Yaskawa INFORM job: A_ROOF_UPPER_0614_2_PAINT_46.JBI

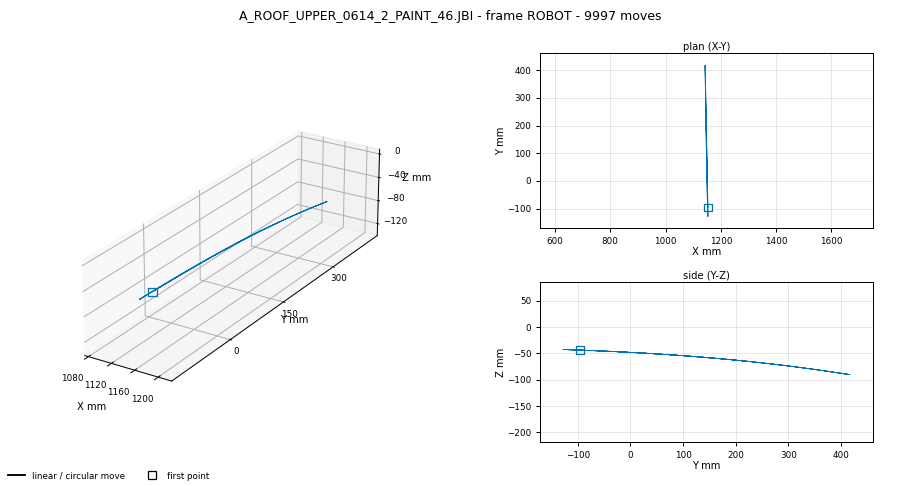
[picture p0: tool path of A_ROOF_UPPER_0614_2_PAINT_46.JBI in frame ROBOT, 9997 of 9997 moves have a stored position in this frame; points joined in program order, loops and branches not executed]
/JOB
//NAME A_ROOF_UPPER_0614_2_PAINT46
//POS
///NPOS 9997,0,0,0,0,0
///TOOL 1
///USER 0
///POSTYPE ROBOT
///RECTAN
///RCONF 1,0,0,0,0,0,0,0,0,0,0,0,0,0,0,0,0,0,0,0,0,0,0,0
C00000=1153.348,-96.269,-43.440,178.853,5.937,149.402
C00001=1153.343,-96.020,-43.449,178.855,5.937,149.401
C00002=1153.337,-95.770,-43.459,178.857,5.937,149.401
C00003=1153.332,-95.520,-43.468,178.859,5.937,149.400
C00004=1153.326,-95.270,-43.478,178.861,5.938,149.400
C00005=1153.321,-95.020,-43.487,178.863,5.939,149.399
C00006=1153.315,-94.771,-43.497,178.865,5.939,149.399
C00007=1153.310,-94.521,-43.506,178.867,5.939,149.398
C00008=1153.304,-94.271,-43.515,178.870,5.940,149.398
C00009=1153.299,-94.021,-43.525,178.871,5.940,149.397
C00010=1153.294,-93.772,-43.534,178.874,5.940,149.396
C00011=1153.289,-93.522,-43.544,178.876,5.941,149.396
C00012=1153.283,-93.272,-43.553,178.878,5.941,149.395
C00013=1153.278,-93.023,-43.563,178.880,5.942,149.395
C00014=1153.273,-92.773,-43.572,178.882,5.941,149.394
C00015=1153.267,-92.523,-43.582,178.884,5.942,149.394
C00016=1153.262,-92.273,-43.592,178.886,5.943,149.393
C00017=1153.257,-92.023,-43.602,178.888,5.942,149.393
C00018=1153.252,-91.773,-43.611,178.891,5.943,149.392
C00019=1153.246,-91.524,-43.621,178.893,5.944,149.392
C00020=1153.241,-91.274,-43.630,178.895,5.943,149.391
C00021=1153.235,-91.024,-43.640,178.897,5.944,149.390
C00022=1153.230,-90.775,-43.649,178.899,5.945,149.390
C00023=1153.225,-90.525,-43.659,178.901,5.945,149.389
C00024=1153.219,-90.275,-43.668,178.904,5.945,149.389
C00025=1153.214,-90.026,-43.678,178.906,5.946,149.388
C00026=1153.209,-89.775,-43.687,178.907,5.946,149.388
C00027=1153.204,-89.526,-43.698,178.910,5.946,149.387
C00028=1153.198,-89.276,-43.707,178.912,5.947,149.387
C00029=1153.193,-89.026,-43.717,178.914,5.947,149.386
C00030=1153.188,-88.777,-43.726,178.917,5.947,149.385
C00031=1153.182,-88.527,-43.736,178.919,5.948,149.385
C00032=1153.176,-88.277,-43.746,178.920,5.948,149.384
C00033=1153.171,-88.027,-43.755,178.923,5.949,149.384
C00034=1153.166,-87.777,-43.766,178.925,5.949,149.383
C00035=1153.161,-87.528,-43.775,178.927,5.949,149.383
C00036=1153.156,-87.278,-43.785,178.929,5.950,149.382
C00037=1153.151,-87.028,-43.794,178.932,5.950,149.382
C00038=1153.145,-86.779,-43.804,178.933,5.950,149.381
C00039=1153.139,-86.529,-43.814,178.935,5.951,149.381
C00040=1153.135,-86.279,-43.824,178.938,5.952,149.380
C00041=1153.129,-86.029,-43.833,178.940,5.952,149.379
C00042=1153.124,-85.779,-43.843,178.942,5.952,149.379
C00043=1153.119,-85.530,-43.853,178.945,5.953,149.378
C00044=1153.113,-85.280,-43.863,178.946,5.953,149.378
C00045=1153.108,-85.031,-43.872,178.948,5.953,149.377
C00046=1153.103,-84.780,-43.883,178.951,5.954,149.377
C00047=1153.098,-84.531,-43.893,178.953,5.954,149.376
C00048=1153.092,-84.281,-43.902,178.955,5.955,149.376
C00049=1153.086,-84.031,-43.912,178.957,5.955,149.375
C00050=1153.082,-83.782,-43.922,178.959,5.955,149.374
C00051=1153.076,-83.531,-43.932,178.961,5.956,149.374
C00052=1153.071,-83.282,-43.942,178.964,5.956,149.373
C00053=1153.066,-83.032,-43.952,178.966,5.956,149.373
C00054=1153.060,-82.783,-43.962,178.968,5.957,149.372
C00055=1153.054,-82.533,-43.971,178.970,5.957,149.372
C00056=1153.050,-82.283,-43.981,178.972,5.957,149.371
C00057=1153.044,-82.033,-43.991,178.974,5.958,149.371
C00058=1153.039,-81.784,-44.002,178.977,5.958,149.370
C00059=1153.034,-81.534,-44.011,178.978,5.958,149.369
C00060=1153.029,-81.284,-44.021,178.981,5.959,149.369
C00061=1153.023,-81.034,-44.031,178.983,5.959,149.368
C00062=1153.017,-80.785,-44.042,178.986,5.960,149.368
C00063=1153.013,-80.535,-44.051,178.987,5.960,149.367
C00064=1153.007,-80.284,-44.061,178.990,5.961,149.366
C00065=1153.002,-80.035,-44.071,178.992,5.961,149.366
C00066=1152.997,-79.786,-44.081,178.994,5.961,149.366
C00067=1152.991,-79.536,-44.091,178.996,5.962,149.365
C00068=1152.986,-79.286,-44.102,178.998,5.962,149.364
C00069=1152.981,-79.036,-44.112,179.000,5.962,149.364
C00070=1152.976,-78.786,-44.121,179.003,5.963,149.363
C00071=1152.970,-78.537,-44.131,179.005,5.964,149.363
C00072=1152.965,-78.287,-44.142,179.008,5.964,149.362
C00073=1152.959,-78.037,-44.152,179.009,5.964,149.361
C00074=1152.954,-77.788,-44.161,179.011,5.965,149.361
C00075=1152.949,-77.538,-44.172,179.014,5.965,149.360
C00076=1152.944,-77.288,-44.182,179.016,5.965,149.360
C00077=1152.938,-77.039,-44.192,179.018,5.966,149.359
C00078=1152.933,-76.767,-44.203,179.020,5.966,149.359
C00079=1152.926,-76.496,-44.214,179.023,5.967,149.358
C00080=1152.921,-76.224,-44.225,179.025,5.967,149.357
C00081=1152.915,-75.953,-44.236,179.028,5.968,149.357
C00082=1152.910,-75.703,-44.246,179.030,5.968,149.356
C00083=1152.905,-75.454,-44.256,179.032,5.969,149.356
C00084=1152.900,-75.204,-44.267,179.034,5.969,149.355
C00085=1152.894,-74.954,-44.277,179.037,5.970,149.355
C00086=1152.888,-74.705,-44.287,179.038,5.970,149.354
C00087=1152.883,-74.455,-44.298,179.041,5.970,149.353
C00088=1152.878,-74.205,-44.308,179.043,5.971,149.353
C00089=1152.872,-73.955,-44.318,179.045,5.971,149.352
C00090=1152.867,-73.706,-44.328,179.047,5.971,149.352
C00091=1152.862,-73.456,-44.338,179.050,5.972,149.351
C00092=1152.857,-73.206,-44.348,179.052,5.972,149.350
C00093=1152.852,-72.956,-44.359,179.054,5.972,149.350
C00094=1152.846,-72.707,-44.369,179.056,5.973,149.350
C00095=1152.841,-72.457,-44.379,179.059,5.974,149.349
C00096=1152.836,-72.207,-44.390,179.061,5.974,149.348
C00097=1152.830,-71.957,-44.400,179.062,5.974,149.348
C00098=1152.825,-71.708,-44.410,179.065,5.975,149.347
C00099=1152.820,-71.458,-44.420,179.067,5.975,149.347
C00100=1152.815,-71.208,-44.431,179.070,5.976,149.346
C00101=1152.809,-70.959,-44.441,179.072,5.976,149.345
C00102=1152.804,-70.708,-44.451,179.074,5.977,149.345
C00103=1152.798,-70.459,-44.462,179.076,5.977,149.344
C00104=1152.793,-70.209,-44.472,179.079,5.978,149.344
C00105=1152.788,-69.960,-44.483,179.080,5.978,149.343
C00106=1152.783,-69.710,-44.493,179.083,5.978,149.343
C00107=1152.778,-69.460,-44.504,179.085,5.979,149.342
C00108=1152.772,-69.210,-44.514,179.088,5.979,149.341
C00109=1152.766,-68.961,-44.524,179.089,5.979,149.341
C00110=1152.761,-68.711,-44.535,179.092,5.980,149.340
C00111=1152.756,-68.461,-44.545,179.094,5.980,149.340
C00112=1152.751,-68.211,-44.556,179.096,5.981,149.339
C00113=1152.745,-67.962,-44.567,179.098,5.981,149.339
C00114=1152.741,-67.713,-44.576,179.101,5.982,149.338
C00115=1152.736,-67.462,-44.587,179.103,5.982,149.338
C00116=1152.730,-67.213,-44.597,179.106,5.983,149.337
C00117=1152.725,-66.963,-44.608,179.107,5.983,149.336
C00118=1152.719,-66.713,-44.618,179.109,5.984,149.336
C00119=1152.715,-66.463,-44.629,179.112,5.984,149.335
C00120=1152.709,-66.214,-44.639,179.114,5.985,149.335
C00121=1152.703,-65.964,-44.649,179.116,5.984,149.334
C00122=1152.698,-65.714,-44.660,179.118,5.985,149.334
C00123=1152.693,-65.465,-44.671,179.121,5.986,149.333
C00124=1152.687,-65.215,-44.682,179.123,5.986,149.332
C00125=1152.682,-64.965,-44.692,179.126,5.987,149.332
C00126=1152.677,-64.715,-44.703,179.128,5.987,149.331
C00127=1152.672,-64.466,-44.714,179.130,5.987,149.331
C00128=1152.667,-64.216,-44.724,179.132,5.988,149.330
C00129=1152.661,-63.966,-44.735,179.135,5.989,149.330
C00130=1152.656,-63.716,-44.745,179.136,5.989,149.329
C00131=1152.651,-63.467,-44.756,179.139,5.989,149.328
C00132=1152.646,-63.217,-44.767,179.141,5.990,149.328
C00133=1152.640,-62.967,-44.777,179.143,5.991,149.327
C00134=1152.635,-62.718,-44.788,179.146,5.991,149.327
C00135=1152.630,-62.468,-44.798,179.148,5.991,149.326
C00136=1152.625,-62.218,-44.809,179.150,5.991,149.326
C00137=1152.620,-61.969,-44.820,179.152,5.992,149.325
C00138=1152.615,-61.719,-44.830,179.155,5.993,149.325
C00139=1152.608,-61.469,-44.841,179.157,5.993,149.324
C00140=1152.603,-61.219,-44.853,179.159,5.993,149.323
C00141=1152.598,-60.970,-44.863,179.162,5.994,149.323
C00142=1152.593,-60.719,-44.873,179.164,5.994,149.322
C00143=1152.588,-60.470,-44.884,179.166,5.995,149.322
C00144=1152.583,-60.220,-44.895,179.169,5.996,149.321
C00145=1152.577,-59.971,-44.906,179.170,5.996,149.321
C00146=1152.572,-59.721,-44.916,179.173,5.996,149.320
C00147=1152.567,-59.472,-44.927,179.175,5.997,149.319
C00148=1152.561,-59.222,-44.938,179.177,5.998,149.319
C00149=1152.556,-58.972,-44.949,179.180,5.998,149.318
C00150=1152.551,-58.722,-44.960,179.181,5.998,149.318
C00151=1152.546,-58.472,-44.970,179.184,5.998,149.317
C00152=1152.541,-58.223,-44.981,179.186,5.999,149.316
C00153=1152.536,-57.973,-44.992,179.188,6.000,149.316
C00154=1152.529,-57.723,-45.003,179.191,6.000,149.315
C00155=1152.525,-57.473,-45.014,179.193,6.000,149.315
C00156=1152.519,-57.224,-45.024,179.195,6.001,149.314
C00157=1152.514,-56.974,-45.036,179.198,6.001,149.314
C00158=1152.509,-56.724,-45.046,179.200,6.002,149.313
C00159=1152.503,-56.475,-45.058,179.202,6.003,149.312
C00160=1152.498,-56.225,-45.068,179.204,6.003,149.312
C00161=1152.493,-55.976,-45.079,179.207,6.003,149.311
C00162=1152.488,-55.725,-45.090,179.209,6.004,149.311
C00163=1152.483,-55.477,-45.101,179.212,6.004,149.310
C00164=1152.477,-55.227,-45.113,179.214,6.005,149.310
C00165=1152.472,-54.976,-45.123,179.216,6.006,149.309
C00166=1152.467,-54.727,-45.134,179.218,6.005,149.308
C00167=1152.462,-54.477,-45.145,179.220,6.006,149.308
C00168=1152.457,-54.227,-45.157,179.223,6.007,149.307
C00169=1152.451,-53.978,-45.167,179.225,6.007,149.307
C00170=1152.446,-53.728,-45.178,179.228,6.008,149.306
C00171=1152.441,-53.479,-45.188,179.230,6.008,149.306
C00172=1152.435,-53.229,-45.200,179.232,6.008,149.305
C00173=1152.431,-52.979,-45.211,179.234,6.009,149.304
C00174=1152.425,-52.729,-45.222,179.236,6.010,149.304
C00175=1152.420,-52.479,-45.233,179.239,6.010,149.303
C00176=1152.415,-52.230,-45.245,179.241,6.011,149.303
C00177=1152.409,-51.980,-45.255,179.243,6.012,149.302
C00178=1152.405,-51.731,-45.266,179.245,6.011,149.302
C00179=1152.398,-51.481,-45.277,179.248,6.012,149.301
C00180=1152.394,-51.231,-45.288,179.250,6.012,149.300
C00181=1152.389,-50.982,-45.300,179.253,6.013,149.300
C00182=1152.383,-50.711,-45.312,179.255,6.014,149.299
C00183=1152.377,-50.440,-45.324,179.257,6.014,149.299
C00184=1152.371,-50.169,-45.336,179.260,6.015,149.298
C00185=1152.365,-49.899,-45.348,179.263,6.015,149.297
C00186=1152.361,-49.649,-45.359,179.265,6.016,149.297
C00187=1152.356,-49.400,-45.371,179.268,6.016,149.296
C00188=1152.350,-49.150,-45.381,179.270,6.017,149.296
C00189=1152.345,-48.900,-45.393,179.271,6.017,149.295
C00190=1152.339,-48.650,-45.405,179.274,6.018,149.294
C00191=1152.334,-48.401,-45.415,179.276,6.018,149.294
C00192=1152.329,-48.151,-45.426,179.279,6.019,149.293
C00193=1152.324,-47.901,-45.438,179.281,6.020,149.293
C00194=1152.319,-47.652,-45.449,179.284,6.020,149.292
C00195=1152.313,-47.402,-45.460,179.286,6.021,149.292
C00196=1152.308,-47.152,-45.471,179.288,6.022,149.291
C00197=1152.303,-46.903,-45.483,179.290,6.021,149.290
C00198=1152.297,-46.653,-45.494,179.292,6.022,149.290
C00199=1152.293,-46.404,-45.505,179.295,6.022,149.289
C00200=1152.287,-46.153,-45.517,179.297,6.023,149.289
C00201=1152.282,-45.904,-45.528,179.300,6.024,149.288
C00202=1152.276,-45.654,-45.539,179.302,6.024,149.288
C00203=1152.271,-45.405,-45.551,179.305,6.025,149.287
C00204=1152.266,-45.155,-45.563,179.307,6.025,149.286
C00205=1152.261,-44.906,-45.573,179.308,6.025,149.286
C00206=1152.256,-44.656,-45.584,179.311,6.026,149.285
C00207=1152.250,-44.406,-45.596,179.313,6.027,149.285
C00208=1152.246,-44.156,-45.607,179.316,6.027,149.284
C00209=1152.240,-43.906,-45.619,179.318,6.028,149.284
C00210=1152.235,-43.657,-45.630,179.321,6.028,149.283
C00211=1152.229,-43.407,-45.642,179.323,6.029,149.282
C00212=1152.225,-43.158,-45.653,179.326,6.029,149.282
C00213=1152.219,-42.908,-45.665,179.327,6.029,149.281
C00214=1152.214,-42.658,-45.675,179.329,6.030,149.281
C00215=1152.208,-42.408,-45.687,179.332,6.031,149.280
C00216=1152.204,-42.159,-45.698,179.334,6.031,149.280
C00217=1152.198,-41.909,-45.710,179.337,6.032,149.279
C00218=1152.193,-41.659,-45.722,179.339,6.033,149.278
C00219=1152.187,-41.410,-45.733,179.342,6.033,149.278
C00220=1152.182,-41.160,-45.745,179.344,6.034,149.277
C00221=1152.177,-40.910,-45.756,179.347,6.034,149.277
C00222=1152.172,-40.660,-45.768,179.349,6.035,149.276
C00223=1152.167,-40.411,-45.779,179.350,6.035,149.276
C00224=1152.161,-40.161,-45.791,179.353,6.035,149.275
C00225=1152.156,-39.912,-45.802,179.355,6.036,149.274
C00226=1152.151,-39.662,-45.814,179.358,6.037,149.274
C00227=1152.146,-39.412,-45.826,179.360,6.037,149.273
C00228=1152.141,-39.162,-45.837,179.363,6.038,149.273
C00229=1152.135,-38.913,-45.849,179.365,6.039,149.272
C00230=1152.130,-38.663,-45.860,179.368,6.039,149.271
C00231=1152.125,-38.413,-45.872,179.370,6.040,149.271
C00232=1152.119,-38.164,-45.884,179.372,6.041,149.270
C00233=1152.115,-37.914,-45.895,179.375,6.041,149.270
C00234=1152.109,-37.664,-45.907,179.377,6.042,149.269
C00235=1152.104,-37.414,-45.918,179.379,6.041,149.269
C00236=1152.099,-37.166,-45.931,179.381,6.042,149.268
C00237=1152.093,-36.916,-45.943,179.384,6.043,149.267
C00238=1152.089,-36.666,-45.954,179.386,6.043,149.267
C00239=1152.083,-36.416,-45.966,179.389,6.044,149.266
C00240=1152.078,-36.166,-45.978,179.391,6.045,149.266
C00241=1152.073,-35.917,-45.989,179.394,6.045,149.265
C00242=1152.068,-35.667,-46.001,179.396,6.046,149.265
C00243=1152.062,-35.417,-46.012,179.398,6.047,149.264
C00244=1152.057,-35.168,-46.024,179.401,6.047,149.263
C00245=1152.052,-34.919,-46.036,179.403,6.048,149.263
C00246=1152.046,-34.669,-46.048,179.405,6.048,149.262
C00247=1152.042,-34.419,-46.059,179.408,6.049,149.262
C00248=1152.036,-34.169,-46.071,179.410,6.050,149.261
C00249=1152.031,-33.919,-46.083,179.412,6.050,149.261
C00250=1152.025,-33.669,-46.095,179.415,6.050,149.260
C00251=1152.021,-33.420,-46.107,179.417,6.051,149.259
C00252=1152.016,-33.170,-46.119,179.419,6.051,149.259
C00253=1152.010,-32.920,-46.131,179.422,6.052,149.258
C00254=1152.005,-32.671,-46.142,179.424,6.053,149.258
C00255=1152.000,-32.422,-46.154,179.426,6.053,149.257
C00256=1151.994,-32.172,-46.166,179.429,6.054,149.257
C00257=1151.989,-31.922,-46.178,179.431,6.054,149.256
C00258=1151.984,-31.673,-46.189,179.433,6.055,149.255
C00259=1151.979,-31.423,-46.202,179.436,6.056,149.255
C00260=1151.974,-31.173,-46.214,179.438,6.056,149.254
C00261=1151.968,-30.923,-46.226,179.441,6.057,149.254
C00262=1151.964,-30.674,-46.237,179.443,6.058,149.253
C00263=1151.958,-30.424,-46.250,179.446,6.058,149.252
C00264=1151.953,-30.174,-46.262,179.448,6.059,149.252
C00265=1151.948,-29.925,-46.273,179.451,6.059,149.251
C00266=1151.942,-29.675,-46.286,179.453,6.060,149.251
C00267=1151.938,-29.426,-46.297,179.455,6.061,149.250
C00268=1151.932,-29.176,-46.309,179.458,6.061,149.250
C00269=1151.927,-28.926,-46.322,179.460,6.062,149.249
C00270=1151.922,-28.676,-46.334,179.463,6.062,149.248
C00271=1151.916,-28.426,-46.346,179.465,6.063,149.248
C00272=1151.911,-28.177,-46.358,179.467,6.064,149.247
C00273=1151.906,-27.928,-46.369,179.469,6.064,149.247
C00274=1151.901,-27.678,-46.381,179.472,6.064,149.246
C00275=1151.896,-27.428,-46.394,179.474,6.065,149.246
C00276=1151.891,-27.178,-46.406,179.476,6.065,149.245
C00277=1151.885,-26.929,-46.418,179.479,6.066,149.244
C00278=1151.880,-26.679,-46.430,179.481,6.067,149.244
C00279=1151.876,-26.430,-46.442,179.483,6.067,149.243
C00280=1151.870,-26.180,-46.454,179.486,6.068,149.243
C00281=1151.865,-25.930,-46.466,179.488,6.069,149.242
C00282=1151.860,-25.681,-46.479,179.490,6.069,149.242
C00283=1151.854,-25.431,-46.491,179.493,6.070,149.241
C00284=1151.849,-25.182,-46.503,179.495,6.071,149.240
C00285=1151.844,-24.932,-46.515,179.498,6.071,149.240
C00286=1151.839,-24.662,-46.529,179.501,6.071,149.239
C00287=1151.833,-24.392,-46.542,179.503,6.073,149.239
C00288=1151.827,-24.122,-46.554,179.506,6.073,149.238
C00289=1151.822,-23.852,-46.569,179.509,6.074,149.237
C00290=1151.816,-23.602,-46.580,179.511,6.075,149.237
C00291=1151.811,-23.353,-46.593,179.513,6.075,149.236
C00292=1151.806,-23.103,-46.605,179.516,6.076,149.236
C00293=1151.801,-22.853,-46.618,179.518,6.077,149.235
C00294=1151.795,-22.603,-46.629,179.521,6.077,149.234
C00295=1151.791,-22.354,-46.641,179.523,6.078,149.234
C00296=1151.785,-22.105,-46.653,179.525,6.078,149.233
C00297=1151.780,-21.855,-46.666,179.528,6.079,149.233
C00298=1151.775,-21.605,-46.678,179.530,6.080,149.232
C00299=1151.770,-21.355,-46.691,179.532,6.080,149.232
C00300=1151.765,-21.106,-46.703,179.535,6.081,149.231
C00301=1151.760,-20.856,-46.715,179.537,6.082,149.230
C00302=1151.755,-20.607,-46.728,179.540,6.082,149.230
C00303=1151.749,-20.357,-46.740,179.542,6.083,149.229
C00304=1151.744,-20.107,-46.752,179.545,6.083,149.229
C00305=1151.738,-19.858,-46.766,179.547,6.084,149.228
C00306=1151.733,-19.608,-46.777,179.550,6.084,149.227
C00307=1151.728,-19.359,-46.790,179.552,6.085,149.227
C00308=1151.723,-19.109,-46.803,179.554,6.086,149.226
C00309=1151.718,-18.859,-46.815,179.557,6.086,149.226
C00310=1151.712,-18.609,-46.827,179.559,6.087,149.225
C00311=1151.707,-18.360,-46.840,179.562,6.088,149.225
C00312=1151.702,-18.110,-46.852,179.564,6.088,149.224
C00313=1151.697,-17.861,-46.865,179.566,6.089,149.223
C00314=1151.692,-17.611,-46.877,179.569,6.090,149.223
C00315=1151.687,-17.361,-46.889,179.571,6.090,149.222
C00316=1151.682,-17.111,-46.902,179.573,6.091,149.222
C00317=1151.677,-16.862,-46.915,179.576,6.091,149.221
C00318=1151.671,-16.613,-46.927,179.579,6.093,149.221
C00319=1151.666,-16.363,-46.939,179.581,6.093,149.220
C00320=1151.661,-16.113,-46.953,179.584,6.094,149.219
C00321=1151.656,-15.863,-46.965,179.586,6.095,149.219
C00322=1151.651,-15.614,-46.978,179.589,6.095,149.218
C00323=1151.645,-15.364,-46.990,179.591,6.096,149.218
C00324=1151.640,-15.115,-47.002,179.593,6.097,149.217
C00325=1151.635,-14.865,-47.015,179.596,6.097,149.216
C00326=1151.630,-14.615,-47.028,179.598,6.098,149.216
C00327=1151.624,-14.366,-47.041,179.600,6.099,149.215
C00328=1151.619,-14.116,-47.054,179.603,6.099,149.215
C00329=1151.614,-13.866,-47.066,179.605,6.100,149.214
C00330=1151.609,-13.616,-47.079,179.608,6.100,149.214
C00331=1151.604,-13.367,-47.091,179.610,6.101,149.213
C00332=1151.599,-13.118,-47.104,179.613,6.102,149.212
C00333=1151.593,-12.868,-47.117,179.615,6.102,149.212
C00334=1151.589,-12.618,-47.130,179.618,6.103,149.211
C00335=1151.583,-12.368,-47.142,179.620,6.104,149.211
C00336=1151.578,-12.119,-47.154,179.622,6.104,149.210
C00337=1151.573,-11.870,-47.167,179.625,6.106,149.210
C00338=1151.568,-11.619,-47.181,179.628,6.106,149.209
C00339=1151.563,-11.370,-47.193,179.630,6.107,149.209
C00340=1151.558,-11.121,-47.206,179.633,6.107,149.208
C00341=1151.552,-10.871,-47.218,179.635,6.108,149.207
C00342=1151.548,-10.621,-47.231,179.637,6.109,149.207
C00343=1151.542,-10.372,-47.245,179.640,6.109,149.206
C00344=1151.537,-10.122,-47.257,179.642,6.110,149.205
C00345=1151.532,-9.873,-47.270,179.644,6.111,149.205
C00346=1151.527,-9.623,-47.283,179.647,6.111,149.205
C00347=1151.521,-9.373,-47.296,179.649,6.112,149.204
C00348=1151.516,-9.124,-47.308,179.652,6.113,149.203
C00349=1151.512,-8.874,-47.321,179.655,6.114,149.203
C00350=1151.507,-8.625,-47.334,179.657,6.115,149.202
C00351=1151.501,-8.375,-47.347,179.660,6.115,149.202
C00352=1151.496,-8.125,-47.360,179.662,6.116,149.201
C00353=1151.491,-7.876,-47.373,179.664,6.116,149.200
C00354=1151.485,-7.626,-47.386,179.667,6.117,149.200
C00355=1151.481,-7.376,-47.399,179.669,6.118,149.199
C00356=1151.476,-7.127,-47.412,179.671,6.118,149.199
C00357=1151.470,-6.877,-47.425,179.674,6.119,149.198
C00358=1151.465,-6.628,-47.437,179.676,6.120,149.198
C00359=1151.460,-6.378,-47.450,179.679,6.120,149.197
C00360=1151.454,-6.128,-47.464,179.682,6.122,149.196
C00361=1151.449,-5.879,-47.476,179.684,6.122,149.196
C00362=1151.445,-5.629,-47.489,179.687,6.123,149.195
C00363=1151.439,-5.380,-47.503,179.689,6.123,149.195
C00364=1151.435,-5.130,-47.516,179.691,6.124,149.194
C00365=1151.429,-4.880,-47.529,179.694,6.125,149.193
C00366=1151.424,-4.631,-47.542,179.696,6.125,149.193
C00367=1151.419,-4.381,-47.555,179.698,6.126,149.193
C00368=1151.413,-4.131,-47.568,179.701,6.127,149.192
C00369=1151.408,-3.882,-47.581,179.704,6.128,149.191
C00370=1151.404,-3.632,-47.594,179.706,6.129,149.191
C00371=1151.398,-3.383,-47.607,179.709,6.130,149.190
C00372=1151.393,-3.133,-47.620,179.711,6.130,149.190
C00373=1151.388,-2.883,-47.634,179.713,6.131,149.189
C00374=1151.382,-2.634,-47.646,179.716,6.131,149.188
C00375=1151.378,-2.384,-47.660,179.718,6.132,149.188
C00376=1151.372,-2.135,-47.673,179.721,6.133,149.187
C00377=1151.368,-1.885,-47.686,179.724,6.134,149.187
C00378=1151.362,-1.635,-47.699,179.726,6.135,149.186
C00379=1151.357,-1.386,-47.712,179.729,6.135,149.186
C00380=1151.352,-1.136,-47.726,179.731,6.136,149.185
C00381=1151.347,-0.887,-47.739,179.733,6.137,149.184
C00382=1151.342,-0.637,-47.752,179.736,6.137,149.184
C00383=1151.337,-0.388,-47.766,179.738,6.138,149.183
C00384=1151.331,-0.138,-47.779,179.741,6.138,149.183
C00385=1151.326,0.112,-47.792,179.744,6.140,149.182
C00386=1151.320,0.361,-47.805,179.746,6.140,149.181
C00387=1151.316,0.611,-47.819,179.748,6.141,149.181
C00388=1151.310,0.860,-47.832,179.751,6.142,149.181
C00389=1151.306,1.110,-47.845,179.753,6.142,149.180
C00390=1151.300,1.379,-47.859,179.757,6.144,149.179
C00391=1151.294,1.649,-47.874,179.759,6.145,149.179
C00392=1151.289,1.918,-47.888,179.761,6.145,149.178
C00393=1151.284,2.188,-47.903,179.765,6.146,149.177
C00394=1151.278,2.437,-47.916,179.767,6.147,149.177
C00395=1151.274,2.687,-47.929,179.769,6.147,149.176
C00396=1151.268,2.936,-47.943,179.772,6.148,149.176
C00397=1151.264,3.186,-47.956,179.774,6.149,149.175
C00398=1151.258,3.435,-47.970,179.776,6.150,149.175
C00399=1151.253,3.686,-47.984,179.779,6.150,149.174
C00400=1151.248,3.935,-47.996,179.782,6.152,149.173
C00401=1151.243,4.185,-48.010,179.784,6.152,149.173
C00402=1151.238,4.434,-48.023,179.787,6.153,149.172
C00403=1151.233,4.684,-48.037,179.789,6.154,149.172
C00404=1151.227,4.933,-48.051,179.792,6.154,149.171
C00405=1151.222,5.183,-48.064,179.794,6.155,149.171
C00406=1151.217,5.432,-48.077,179.797,6.156,149.170
C00407=1151.212,5.682,-48.091,179.799,6.157,149.169
C00408=1151.207,5.932,-48.104,179.802,6.157,149.169
C00409=1151.202,6.181,-48.119,179.804,6.158,149.168
C00410=1151.196,6.431,-48.131,179.807,6.159,149.168
C00411=1151.192,6.680,-48.145,179.809,6.160,149.167
C00412=1151.186,6.930,-48.159,179.812,6.161,149.166
C00413=1151.181,7.179,-48.172,179.814,6.162,149.166
C00414=1151.176,7.430,-48.186,179.817,6.162,149.165
C00415=1151.171,7.679,-48.200,179.819,6.163,149.165
C00416=1151.166,7.928,-48.213,179.822,6.163,149.164
C00417=1151.161,8.178,-48.227,179.824,6.165,149.164
C00418=1151.156,8.427,-48.241,179.827,6.166,149.163
C00419=1151.150,8.677,-48.254,179.829,6.166,149.163
C00420=1151.146,8.926,-48.268,179.831,6.167,149.162
C00421=1151.141,9.176,-48.282,179.834,6.167,149.161
C00422=1151.135,9.426,-48.295,179.837,6.169,149.161
C00423=1151.130,9.675,-48.309,179.840,6.170,149.160
C00424=1151.125,9.925,-48.322,179.842,6.170,149.160
C00425=1151.120,10.174,-48.336,179.844,6.171,149.159
C00426=1151.115,10.424,-48.350,179.847,6.172,149.159
C00427=1151.110,10.674,-48.363,179.850,6.173,149.158
C00428=1151.105,10.923,-48.378,179.852,6.174,149.158
C00429=1151.099,11.172,-48.392,179.855,6.174,149.157
C00430=1151.094,11.423,-48.405,179.857,6.175,149.156
C00431=1151.090,11.672,-48.419,179.860,6.176,149.156
C00432=1151.084,11.921,-48.433,179.862,6.177,149.155
C00433=1151.079,12.171,-48.447,179.864,6.178,149.155
C00434=1151.074,12.421,-48.461,179.867,6.178,149.154
C00435=1151.069,12.670,-48.474,179.869,6.179,149.154
C00436=1151.064,12.919,-48.488,179.872,6.180,149.153
C00437=1151.058,13.169,-48.501,179.875,6.181,149.153
C00438=1151.053,13.419,-48.516,179.877,6.182,149.152
C00439=1151.048,13.668,-48.530,179.879,6.182,149.151
C00440=1151.043,13.917,-48.544,179.883,6.184,149.151
C00441=1151.038,14.167,-48.557,179.885,6.185,149.150
C00442=1151.033,14.417,-48.571,179.888,6.185,149.150
C00443=1151.028,14.666,-48.585,179.890,6.186,149.149
C00444=1151.023,14.916,-48.599,179.892,6.186,149.148
C00445=1151.018,15.166,-48.613,179.895,6.188,149.148
C00446=1151.013,15.415,-48.628,179.898,6.188,149.147
C00447=1151.007,15.665,-48.641,179.900,6.189,149.147
C00448=1151.003,15.914,-48.655,179.902,6.190,149.146
C00449=1150.998,16.164,-48.669,179.905,6.191,149.146
C00450=1150.992,16.413,-48.683,179.907,6.192,149.145
C00451=1150.987,16.663,-48.697,179.910,6.193,149.145
C00452=1150.982,16.913,-48.711,179.912,6.193,149.144
C00453=1150.977,17.162,-48.726,179.916,6.195,149.143
C00454=1150.972,17.411,-48.740,179.918,6.195,149.143
C00455=1150.967,17.661,-48.754,179.920,6.196,149.142
C00456=1150.962,17.911,-48.767,179.923,6.197,149.142
C00457=1150.956,18.160,-48.781,179.926,6.198,149.141
C00458=1150.951,18.410,-48.796,179.928,6.199,149.141
C00459=1150.946,18.660,-48.810,179.931,6.199,149.140
C00460=1150.942,18.909,-48.824,179.933,6.200,149.140
C00461=1150.936,19.158,-48.837,179.936,6.202,149.139
C00462=1150.931,19.408,-48.852,179.938,6.202,149.138
C00463=1150.926,19.658,-48.866,179.940,6.203,149.138
C00464=1150.921,19.907,-48.880,179.943,6.203,149.137
C00465=1150.916,20.156,-48.894,179.946,6.205,149.137
C00466=1150.911,20.406,-48.909,179.948,6.206,149.136
C00467=1150.906,20.656,-48.923,179.951,6.206,149.136
C00468=1150.901,20.905,-48.937,179.954,6.208,149.135
C00469=1150.896,21.155,-48.951,179.956,6.208,149.134
C00470=1150.891,21.404,-48.965,179.959,6.209,149.134
C00471=1150.886,21.654,-48.980,179.961,6.210,149.133
C00472=1150.881,21.904,-48.994,179.964,6.211,149.133
C00473=1150.876,22.153,-49.008,179.966,6.212,149.132
C00474=1150.870,22.403,-49.024,179.968,6.213,149.132
C00475=1150.865,22.652,-49.038,179.971,6.213,149.131
C00476=1150.860,22.901,-49.052,179.974,6.215,149.131
C00477=1150.855,23.151,-49.066,179.976,6.215,149.130
C00478=1150.850,23.401,-49.080,179.979,6.216,149.129
C00479=1150.845,23.650,-49.095,179.982,6.217,149.129
C00480=1150.840,23.900,-49.109,179.984,6.218,149.128
C00481=1150.834,24.149,-49.123,179.987,6.219,149.128
C00482=1150.829,24.399,-49.137,179.989,6.220,149.127
C00483=1150.825,24.648,-49.152,179.992,6.221,149.127
C00484=1150.820,24.898,-49.166,179.994,6.221,149.126
C00485=1150.815,25.147,-49.181,179.996,6.222,149.126
C00486=1150.809,25.397,-49.196,180.000,6.224,149.125
C00487=1150.804,25.646,-49.209,-179.998,6.224,149.125
C00488=1150.799,25.896,-49.224,-179.996,6.225,149.124
C00489=1150.794,26.145,-49.239,-179.993,6.226,149.123
C00490=1150.789,26.395,-49.253,-179.990,6.227,149.123
C00491=1150.784,26.645,-49.267,-179.988,6.228,149.122
C00492=1150.779,26.894,-49.282,-179.985,6.229,149.122
C00493=1150.774,27.144,-49.297,-179.983,6.230,149.121
C00494=1150.769,27.413,-49.313,-179.980,6.230,149.120
C00495=1150.763,27.682,-49.328,-179.977,6.232,149.120
C00496=1150.758,27.950,-49.343,-179.974,6.232,149.119
C00497=1150.752,28.219,-49.360,-179.971,6.234,149.119
C00498=1150.747,28.469,-49.374,-179.969,6.234,149.118
C00499=1150.742,28.719,-49.388,-179.966,6.236,149.118
C00500=1150.737,28.968,-49.403,-179.964,6.237,149.117
C00501=1150.732,29.217,-49.417,-179.961,6.237,149.117
C00502=1150.726,29.467,-49.432,-179.959,6.238,149.116
C00503=1150.722,29.717,-49.447,-179.956,6.240,149.115
C00504=1150.717,29.966,-49.461,-179.953,6.240,149.115
C00505=1150.712,30.216,-49.476,-179.951,6.241,149.114
C00506=1150.706,30.465,-49.491,-179.948,6.242,149.114
C00507=1150.702,30.715,-49.506,-179.946,6.243,149.113
C00508=1150.697,30.964,-49.521,-179.944,6.244,149.113
C00509=1150.692,31.214,-49.535,-179.940,6.245,149.112
C00510=1150.686,31.463,-49.549,-179.938,6.246,149.112
C00511=1150.681,31.712,-49.564,-179.935,6.247,149.111
C00512=1150.676,31.962,-49.579,-179.933,6.248,149.110
C00513=1150.671,32.211,-49.594,-179.930,6.248,149.110
C00514=1150.666,32.461,-49.609,-179.927,6.250,149.109
C00515=1150.661,32.710,-49.624,-179.925,6.251,149.109
C00516=1150.656,32.960,-49.638,-179.923,6.251,149.108
C00517=1150.651,33.209,-49.653,-179.920,6.253,149.108
C00518=1150.646,33.459,-49.668,-179.917,6.253,149.107
C00519=1150.641,33.708,-49.683,-179.915,6.254,149.107
C00520=1150.635,33.958,-49.698,-179.912,6.256,149.106
C00521=1150.631,34.207,-49.713,-179.910,6.256,149.106
C00522=1150.625,34.457,-49.727,-179.907,6.257,149.105
C00523=1150.620,34.706,-49.742,-179.904,6.259,149.104
C00524=1150.615,34.956,-49.757,-179.902,6.259,149.104
C00525=1150.610,35.205,-49.772,-179.900,6.260,149.103
C00526=1150.605,35.455,-49.787,-179.897,6.261,149.103
C00527=1150.600,35.704,-49.802,-179.894,6.262,149.102
C00528=1150.595,35.954,-49.816,-179.891,6.264,149.102
C00529=1150.591,36.204,-49.832,-179.889,6.264,149.101
C00530=1150.585,36.453,-49.847,-179.887,6.265,149.101
C00531=1150.580,36.703,-49.862,-179.883,6.266,149.100
C00532=1150.576,36.952,-49.877,-179.881,6.267,149.099
C00533=1150.570,37.202,-49.891,-179.879,6.268,149.099
C00534=1150.565,37.451,-49.906,-179.876,6.269,149.098
C00535=1150.560,37.701,-49.922,-179.874,6.270,149.098
C00536=1150.555,37.950,-49.936,-179.870,6.271,149.097
C00537=1150.550,38.200,-49.952,-179.868,6.272,149.097
C00538=1150.545,38.449,-49.967,-179.866,6.272,149.096
C00539=1150.539,38.699,-49.982,-179.863,6.274,149.096
C00540=1150.535,38.948,-49.997,-179.861,6.275,149.095
C00541=1150.529,39.197,-50.012,-179.857,6.276,149.095
C00542=1150.524,39.447,-50.027,-179.855,6.277,149.094
C00543=1150.520,39.696,-50.042,-179.853,6.278,149.093
C00544=1150.515,39.946,-50.058,-179.850,6.279,149.093
C00545=1150.510,40.195,-50.073,-179.847,6.280,149.092
C00546=1150.505,40.446,-50.087,-179.844,6.281,149.092
C00547=1150.499,40.695,-50.103,-179.842,6.282,149.091
C00548=1150.495,40.944,-50.118,-179.840,6.283,149.091
C00549=1150.489,41.193,-50.134,-179.837,6.284,149.090
C00550=1150.484,41.443,-50.148,-179.834,6.285,149.090
C00551=1150.479,41.693,-50.163,-179.831,6.286,149.089
C00552=1150.475,41.942,-50.179,-179.829,6.287,149.089
C00553=1150.469,42.192,-50.194,-179.827,6.288,149.088
C00554=1150.465,42.441,-50.209,-179.824,6.289,149.088
C00555=1150.459,42.691,-50.224,-179.821,6.290,149.087
C00556=1150.454,42.940,-50.239,-179.818,6.291,149.086
C00557=1150.449,43.189,-50.255,-179.816,6.292,149.086
C00558=1150.444,43.439,-50.271,-179.813,6.294,149.085
C00559=1150.440,43.689,-50.286,-179.811,6.294,149.085
C00560=1150.434,43.938,-50.301,-179.808,6.295,149.084
C00561=1150.429,44.188,-50.316,-179.806,6.297,149.084
C00562=1150.424,44.437,-50.331,-179.803,6.297,149.083
C00563=1150.418,44.686,-50.347,-179.800,6.299,149.083
C00564=1150.414,44.936,-50.362,-179.798,6.300,149.082
C00565=1150.409,45.186,-50.378,-179.795,6.301,149.082
C00566=1150.404,45.435,-50.393,-179.793,6.302,149.081
C00567=1150.399,45.684,-50.408,-179.790,6.302,149.080
C00568=1150.394,45.934,-50.424,-179.787,6.304,149.080
C00569=1150.390,46.183,-50.439,-179.785,6.304,149.079
C00570=1150.384,46.433,-50.455,-179.782,6.306,149.079
C00571=1150.379,46.682,-50.471,-179.780,6.307,149.078
C00572=1150.374,46.931,-50.486,-179.776,6.308,149.078
C00573=1150.369,47.181,-50.501,-179.774,6.309,149.077
C00574=1150.364,47.431,-50.517,-179.772,6.309,149.077
C00575=1150.359,47.680,-50.533,-179.769,6.311,149.076
C00576=1150.354,47.929,-50.548,-179.767,6.312,149.076
C00577=1150.349,48.179,-50.564,-179.763,6.313,149.075
C00578=1150.344,48.429,-50.579,-179.761,6.314,149.075
C00579=1150.339,48.678,-50.594,-179.758,6.315,149.074
C00580=1150.334,48.927,-50.610,-179.756,6.316,149.074
C00581=1150.329,49.177,-50.626,-179.753,6.318,149.073
C00582=1150.324,49.427,-50.641,-179.751,6.318,149.072
C00583=1150.319,49.676,-50.656,-179.748,6.320,149.072
C00584=1150.313,49.925,-50.672,-179.745,6.320,149.071
C00585=1150.309,50.175,-50.689,-179.742,6.322,149.071
C00586=1150.304,50.424,-50.704,-179.740,6.323,149.070
C00587=1150.299,50.673,-50.719,-179.738,6.323,149.070
C00588=1150.294,50.923,-50.735,-179.735,6.325,149.069
C00589=1150.289,51.173,-50.751,-179.732,6.325,149.069
C00590=1150.283,51.422,-50.766,-179.729,6.327,149.068
C00591=1150.279,51.672,-50.782,-179.727,6.328,149.068
C00592=1150.274,51.921,-50.798,-179.724,6.329,149.067
C00593=1150.269,52.170,-50.814,-179.722,6.330,149.067
C00594=1150.264,52.420,-50.829,-179.719,6.331,149.066
C00595=1150.259,52.670,-50.845,-179.717,6.332,149.066
C00596=1150.253,52.919,-50.861,-179.714,6.334,149.065
C00597=1150.250,53.168,-50.877,-179.711,6.334,149.064
C00598=1150.244,53.437,-50.894,-179.708,6.336,149.064
C00599=1150.238,53.705,-50.911,-179.705,6.337,149.063
C00600=1150.233,53.974,-50.928,-179.703,6.338,149.063
C00601=1150.227,54.242,-50.945,-179.700,6.339,149.062
C00602=1150.223,54.492,-50.961,-179.697,6.341,149.062
C00603=1150.217,54.742,-50.976,-179.694,6.342,149.061
C00604=1150.212,54.991,-50.992,-179.692,6.343,149.061
C00605=1150.207,55.240,-51.009,-179.689,6.344,149.060
C00606=1150.202,55.490,-51.024,-179.686,6.345,149.060
C00607=1150.197,55.739,-51.040,-179.684,6.346,149.059
C00608=1150.193,55.988,-51.056,-179.681,6.347,149.058
C00609=1150.187,56.238,-51.071,-179.679,6.348,149.058
C00610=1150.183,56.488,-51.087,-179.676,6.350,149.058
C00611=1150.178,56.737,-51.104,-179.673,6.350,149.057
C00612=1150.172,56.986,-51.119,-179.671,6.352,149.056
C00613=1150.167,57.236,-51.135,-179.668,6.353,149.056
C00614=1150.162,57.485,-51.152,-179.665,6.354,149.055
C00615=1150.158,57.735,-51.167,-179.663,6.355,149.055
C00616=1150.152,57.984,-51.184,-179.660,6.356,149.054
C00617=1150.148,58.234,-51.200,-179.658,6.357,149.054
C00618=1150.142,58.483,-51.215,-179.654,6.359,149.053
C00619=1150.137,58.732,-51.232,-179.652,6.359,149.053
C00620=1150.132,58.982,-51.248,-179.649,6.361,149.052
C00621=1150.127,59.231,-51.264,-179.647,6.362,149.052
C00622=1150.123,59.481,-51.280,-179.644,6.363,149.051
C00623=1150.117,59.730,-51.296,-179.642,6.364,149.051
C00624=1150.113,59.980,-51.312,-179.639,6.365,149.050
C00625=1150.108,60.229,-51.328,-179.637,6.366,149.050
C00626=1150.103,60.479,-51.344,-179.634,6.368,149.049
C00627=1150.098,60.728,-51.361,-179.631,6.368,149.049
C00628=1150.093,60.978,-51.377,-179.628,6.370,149.048
C00629=1150.088,61.227,-51.393,-179.625,6.371,149.047
C00630=1150.083,61.477,-51.409,-179.623,6.372,149.047
C00631=1150.078,61.726,-51.425,-179.620,6.374,149.047
C00632=1150.072,61.975,-51.442,-179.618,6.374,149.046
C00633=1150.067,62.225,-51.458,-179.615,6.376,149.045
C00634=1150.062,62.473,-51.474,-179.613,6.377,149.045
C00635=1150.058,62.724,-51.490,-179.610,6.378,149.044
C00636=1150.053,62.973,-51.507,-179.607,6.379,149.044
C00637=1150.048,63.222,-51.523,-179.605,6.381,149.043
C00638=1150.043,63.472,-51.539,-179.601,6.382,149.043
C00639=1150.038,63.721,-51.556,-179.599,6.383,149.042
C00640=1150.033,63.971,-51.571,-179.596,6.384,149.042
C00641=1150.027,64.220,-51.588,-179.594,6.385,149.041
C00642=1150.023,64.469,-51.605,-179.591,6.387,149.041
C00643=1150.018,64.719,-51.621,-179.589,6.387,149.040
C00644=1150.013,64.968,-51.637,-179.586,6.389,149.040
C00645=1150.008,65.217,-51.654,-179.583,6.390,149.039
C00646=1150.003,65.467,-51.670,-179.580,6.391,149.039
C00647=1149.997,65.716,-51.686,-179.578,6.392,149.038
C00648=1149.993,65.966,-51.703,-179.575,6.393,149.038
C00649=1149.988,66.215,-51.720,-179.572,6.395,149.037
C00650=1149.983,66.465,-51.735,-179.570,6.396,149.037
C00651=1149.979,66.714,-51.752,-179.567,6.397,149.036
C00652=1149.973,66.963,-51.769,-179.564,6.398,149.036
C00653=1149.968,67.213,-51.786,-179.562,6.399,149.035
C00654=1149.964,67.463,-51.802,-179.559,6.401,149.035
C00655=1149.958,67.712,-51.818,-179.557,6.401,149.034
C00656=1149.954,67.961,-51.835,-179.554,6.403,149.034
C00657=1149.948,68.210,-51.851,-179.551,6.404,149.033
C00658=1149.944,68.460,-51.868,-179.548,6.405,149.033
C00659=1149.939,68.709,-51.885,-179.546,6.407,149.032
C00660=1149.934,68.959,-51.900,-179.543,6.407,149.031
C00661=1149.929,69.208,-51.918,-179.540,6.409,149.031
C00662=1149.924,69.458,-51.934,-179.538,6.410,149.031
C00663=1149.919,69.707,-51.951,-179.535,6.411,149.030
C00664=1149.914,69.956,-51.968,-179.532,6.413,149.029
C00665=1149.909,70.205,-51.984,-179.530,6.414,149.029
C00666=1149.904,70.455,-52.001,-179.527,6.415,149.028
C00667=1149.899,70.704,-52.018,-179.524,6.417,149.028
C00668=1149.894,70.954,-52.034,-179.522,6.418,149.028
C00669=1149.889,71.203,-52.050,-179.519,6.419,149.027
C00670=1149.884,71.453,-52.068,-179.517,6.420,149.026
C00671=1149.879,71.702,-52.084,-179.514,6.421,149.026
C00672=1149.874,71.951,-52.101,-179.511,6.423,149.025
C00673=1149.869,72.201,-52.118,-179.508,6.424,149.025
C00674=1149.864,72.450,-52.134,-179.506,6.425,149.024
C00675=1149.860,72.700,-52.151,-179.503,6.426,149.024
C00676=1149.854,72.949,-52.168,-179.500,6.427,149.023
C00677=1149.850,73.199,-52.185,-179.498,6.429,149.023
C00678=1149.844,73.448,-52.202,-179.495,6.430,149.023
C00679=1149.840,73.697,-52.218,-179.492,6.431,149.022
C00680=1149.835,73.947,-52.235,-179.490,6.433,149.021
C00681=1149.829,74.196,-52.252,-179.487,6.434,149.021
C00682=1149.825,74.445,-52.269,-179.484,6.435,149.020
C00683=1149.820,74.695,-52.287,-179.481,6.437,149.020
C00684=1149.815,74.944,-52.303,-179.479,6.438,149.020
C00685=1149.810,75.193,-52.320,-179.476,6.439,149.019
C00686=1149.805,75.443,-52.337,-179.474,6.440,149.018
C00687=1149.801,75.692,-52.353,-179.471,6.441,149.018
C00688=1149.795,75.941,-52.370,-179.468,6.443,149.017
C00689=1149.790,76.191,-52.387,-179.466,6.444,149.017
C00690=1149.785,76.441,-52.404,-179.463,6.445,149.016
C00691=1149.781,76.690,-52.421,-179.460,6.447,149.016
C00692=1149.776,76.939,-52.439,-179.458,6.447,149.015
C00693=1149.771,77.188,-52.455,-179.455,6.449,149.015
C00694=1149.765,77.438,-52.472,-179.452,6.450,149.014
C00695=1149.761,77.687,-52.489,-179.450,6.451,149.014
C00696=1149.756,77.937,-52.506,-179.447,6.453,149.013
C00697=1149.751,78.185,-52.523,-179.444,6.455,149.013
C00698=1149.746,78.435,-52.541,-179.441,6.455,149.012
C00699=1149.741,78.684,-52.557,-179.439,6.457,149.012
C00700=1149.736,78.934,-52.575,-179.436,6.459,149.012
C00701=1149.731,79.183,-52.593,-179.433,6.459,149.011
C00702=1149.726,79.451,-52.610,-179.431,6.461,149.010
C00703=1149.721,79.720,-52.629,-179.427,6.462,149.010
C00704=1149.715,79.988,-52.647,-179.425,6.464,149.009
C00705=1149.710,80.257,-52.665,-179.421,6.465,149.009
C00706=1149.705,80.507,-52.683,-179.419,6.467,149.008
C00707=1149.700,80.756,-52.700,-179.417,6.467,149.008
C00708=1149.695,81.005,-52.717,-179.414,6.469,149.007
C00709=1149.689,81.254,-52.734,-179.411,6.470,149.007
C00710=1149.685,81.503,-52.752,-179.408,6.471,149.006
C00711=1149.680,81.753,-52.769,-179.406,6.473,149.006
C00712=1149.676,82.003,-52.786,-179.402,6.474,149.005
C00713=1149.671,82.252,-52.804,-179.400,6.475,149.005
C00714=1149.665,82.502,-52.821,-179.398,6.477,149.004
C00715=1149.661,82.750,-52.838,-179.395,6.479,149.004
C00716=1149.656,83.000,-52.856,-179.392,6.479,149.003
C00717=1149.650,83.249,-52.872,-179.389,6.481,149.003
C00718=1149.646,83.498,-52.890,-179.387,6.482,149.003
C00719=1149.641,83.748,-52.907,-179.384,6.484,149.002
C00720=1149.636,83.997,-52.925,-179.381,6.485,149.001
C00721=1149.631,84.247,-52.942,-179.379,6.486,149.001
C00722=1149.627,84.496,-52.960,-179.376,6.488,149.001
C00723=1149.621,84.746,-52.977,-179.373,6.488,149.000
C00724=1149.616,84.995,-52.995,-179.371,6.490,148.999
C00725=1149.612,85.244,-53.012,-179.368,6.492,148.999
C00726=1149.607,85.493,-53.030,-179.365,6.493,148.998
C00727=1149.601,85.743,-53.046,-179.362,6.494,148.998
C00728=1149.596,85.992,-53.064,-179.360,6.496,148.998
C00729=1149.592,86.241,-53.081,-179.357,6.497,148.997
C00730=1149.587,86.490,-53.099,-179.354,6.498,148.997
C00731=1149.582,86.740,-53.116,-179.352,6.500,148.996
C00732=1149.577,86.989,-53.134,-179.349,6.501,148.996
C00733=1149.573,87.238,-53.152,-179.346,6.503,148.995
C00734=1149.567,87.488,-53.169,-179.344,6.503,148.995
C00735=1149.562,87.737,-53.187,-179.341,6.505,148.994
C00736=1149.557,87.987,-53.204,-179.338,6.507,148.994
C00737=1149.552,88.236,-53.222,-179.336,6.508,148.993
C00738=1149.548,88.485,-53.240,-179.333,6.509,148.993
C00739=1149.543,88.735,-53.257,-179.330,6.511,148.992
C00740=1149.538,88.984,-53.275,-179.327,6.512,148.992
C00741=1149.533,89.233,-53.293,-179.325,6.513,148.991
C00742=1149.528,89.483,-53.310,-179.322,6.514,148.991
C00743=1149.523,89.732,-53.328,-179.319,6.516,148.990
C00744=1149.519,89.981,-53.345,-179.316,6.518,148.990
C00745=1149.514,90.231,-53.363,-179.314,6.518,148.989
C00746=1149.509,90.480,-53.381,-179.311,6.520,148.989
C00747=1149.504,90.729,-53.399,-179.308,6.522,148.988
C00748=1149.499,90.978,-53.417,-179.306,6.523,148.988
C00749=1149.494,91.228,-53.434,-179.303,6.524,148.987
C00750=1149.489,91.477,-53.452,-179.300,6.526,148.987
C00751=1149.484,91.726,-53.470,-179.297,6.527,148.987
C00752=1149.479,91.976,-53.488,-179.295,6.529,148.986
C00753=1149.474,92.225,-53.505,-179.292,6.530,148.985
C00754=1149.470,92.474,-53.523,-179.289,6.531,148.985
C00755=1149.465,92.723,-53.540,-179.287,6.533,148.985
C00756=1149.460,92.973,-53.558,-179.284,6.534,148.984
C00757=1149.455,93.223,-53.577,-179.281,6.536,148.984
C00758=1149.450,93.472,-53.595,-179.279,6.537,148.983
C00759=1149.445,93.722,-53.612,-179.276,6.538,148.983
C00760=1149.440,93.971,-53.630,-179.273,6.540,148.982
C00761=1149.435,94.220,-53.648,-179.270,6.542,148.982
C00762=1149.431,94.469,-53.666,-179.268,6.542,148.981
C00763=1149.426,94.718,-53.684,-179.265,6.544,148.981
C00764=1149.421,94.967,-53.702,-179.262,6.546,148.980
C00765=1149.416,95.217,-53.720,-179.260,6.547,148.980
C00766=1149.411,95.466,-53.738,-179.256,6.549,148.979
C00767=1149.406,95.715,-53.756,-179.254,6.549,148.979
C00768=1149.402,95.965,-53.774,-179.251,6.551,148.978
C00769=1149.396,96.215,-53.792,-179.249,6.553,148.978
C00770=1149.391,96.464,-53.809,-179.246,6.555,148.978
C00771=1149.387,96.713,-53.827,-179.243,6.556,148.977
C00772=1149.381,96.962,-53.846,-179.241,6.557,148.977
C00773=1149.376,97.212,-53.864,-179.238,6.558,148.976
C00774=1149.371,97.461,-53.882,-179.235,6.560,148.976
C00775=1149.367,97.711,-53.900,-179.232,6.561,148.975
C00776=1149.362,97.960,-53.918,-179.229,6.563,148.975
C00777=1149.357,98.208,-53.937,-179.227,6.564,148.974
C00778=1149.352,98.458,-53.955,-179.224,6.566,148.974
C00779=1149.347,98.707,-53.973,-179.222,6.567,148.973
C00780=1149.343,98.956,-53.991,-179.218,6.569,148.973
C00781=1149.338,99.206,-54.009,-179.216,6.570,148.972
C00782=1149.333,99.455,-54.028,-179.214,6.571,148.972
C00783=1149.328,99.704,-54.046,-179.211,6.573,148.972
C00784=1149.323,99.954,-54.064,-179.208,6.575,148.971
C00785=1149.318,100.203,-54.082,-179.205,6.576,148.971
C00786=1149.314,100.453,-54.100,-179.202,6.578,148.970
C00787=1149.309,100.701,-54.119,-179.199,6.579,148.970
C00788=1149.304,100.950,-54.137,-179.197,6.580,148.969
C00789=1149.298,101.200,-54.155,-179.195,6.582,148.969
C00790=1149.293,101.449,-54.173,-179.191,6.583,148.968
C00791=1149.289,101.699,-54.192,-179.189,6.585,148.968
C00792=1149.284,101.948,-54.210,-179.186,6.587,148.967
C00793=1149.280,102.197,-54.228,-179.183,6.588,148.967
C00794=1149.274,102.446,-54.247,-179.181,6.589,148.967
C00795=1149.270,102.696,-54.265,-179.178,6.590,148.966
C00796=1149.265,102.945,-54.283,-179.175,6.592,148.966
C00797=1149.260,103.194,-54.302,-179.172,6.594,148.965
C00798=1149.255,103.443,-54.321,-179.170,6.596,148.965
C00799=1149.250,103.693,-54.339,-179.167,6.597,148.964
C00800=1149.245,103.942,-54.357,-179.164,6.599,148.964
C00801=1149.241,104.191,-54.376,-179.162,6.599,148.963
C00802=1149.235,104.440,-54.394,-179.159,6.601,148.963
C00803=1149.231,104.690,-54.413,-179.156,6.603,148.962
C00804=1149.226,104.939,-54.431,-179.153,6.604,148.962
C00805=1149.220,105.188,-54.450,-179.151,6.606,148.962
C00806=1149.216,105.457,-54.470,-179.147,6.608,148.961
C00807=1149.210,105.726,-54.490,-179.145,6.609,148.961
C00808=1149.205,105.993,-54.510,-179.141,6.611,148.960
C00809=1149.200,106.262,-54.530,-179.139,6.612,148.959
C00810=1149.195,106.512,-54.548,-179.136,6.614,148.959
C00811=1149.191,106.760,-54.567,-179.133,6.616,148.959
C00812=1149.185,107.010,-54.585,-179.131,6.617,148.958
C00813=1149.180,107.258,-54.604,-179.127,6.619,148.958
C00814=1149.176,107.508,-54.622,-179.125,6.620,148.957
C00815=1149.171,107.757,-54.642,-179.123,6.621,148.957
C00816=1149.166,108.007,-54.660,-179.120,6.623,148.956
C00817=1149.162,108.256,-54.679,-179.117,6.625,148.956
C00818=1149.156,108.505,-54.697,-179.114,6.626,148.956
C00819=1149.152,108.755,-54.716,-179.112,6.628,148.955
C00820=1149.147,109.004,-54.735,-179.108,6.629,148.955
C00821=1149.142,109.253,-54.753,-179.106,6.631,148.954
C00822=1149.137,109.503,-54.773,-179.103,6.633,148.954
C00823=1149.132,109.751,-54.791,-179.101,6.634,148.953
C00824=1149.128,110.001,-54.810,-179.098,6.635,148.953
C00825=1149.123,110.250,-54.829,-179.095,6.637,148.952
C00826=1149.118,110.499,-54.847,-179.092,6.638,148.952
C00827=1149.113,110.749,-54.867,-179.089,6.640,148.951
C00828=1149.108,110.998,-54.884,-179.087,6.642,148.951
C00829=1149.103,111.247,-54.904,-179.084,6.643,148.951
C00830=1149.099,111.496,-54.923,-179.081,6.645,148.950
C00831=1149.093,111.745,-54.941,-179.079,6.647,148.950
C00832=1149.089,111.995,-54.960,-179.076,6.648,148.949
C00833=1149.083,112.244,-54.979,-179.073,6.650,148.949
C00834=1149.079,112.493,-54.998,-179.070,6.651,148.948
C00835=1149.074,112.742,-55.017,-179.068,6.652,148.948
C00836=1149.069,112.992,-55.035,-179.065,6.654,148.948
C00837=1149.064,113.241,-55.055,-179.062,6.656,148.947
C00838=1149.059,113.490,-55.074,-179.060,6.657,148.947
C00839=1149.055,113.739,-55.093,-179.057,6.659,148.946
C00840=1149.049,113.989,-55.112,-179.054,6.660,148.946
C00841=1149.045,114.238,-55.131,-179.051,6.662,148.945
C00842=1149.040,114.487,-55.150,-179.048,6.664,148.945
C00843=1149.036,114.737,-55.169,-179.045,6.666,148.944
C00844=1149.030,114.986,-55.188,-179.043,6.667,148.944
C00845=1149.026,115.235,-55.208,-179.040,6.669,148.944
C00846=1149.021,115.484,-55.226,-179.037,6.671,148.943
C00847=1149.016,115.733,-55.246,-179.035,6.672,148.943
C00848=1149.011,115.982,-55.264,-179.032,6.673,148.942
C00849=1149.007,116.232,-55.284,-179.029,6.675,148.942
C00850=1149.001,116.481,-55.303,-179.027,6.676,148.941
C00851=1148.997,116.730,-55.322,-179.024,6.678,148.941
C00852=1148.992,116.979,-55.341,-179.021,6.680,148.941
C00853=1148.987,117.229,-55.361,-179.018,6.681,148.940
C00854=1148.982,117.478,-55.379,-179.016,6.683,148.940
C00855=1148.978,117.727,-55.399,-179.013,6.685,148.939
C00856=1148.972,117.976,-55.418,-179.010,6.686,148.939
C00857=1148.968,118.225,-55.437,-179.007,6.688,148.939
C00858=1148.963,118.474,-55.456,-179.004,6.690,148.938
C00859=1148.958,118.724,-55.476,-179.002,6.691,148.938
C00860=1148.953,118.973,-55.495,-178.999,6.693,148.937
C00861=1148.949,119.222,-55.514,-178.996,6.695,148.937
C00862=1148.944,119.472,-55.534,-178.993,6.696,148.936
C00863=1148.939,119.720,-55.553,-178.991,6.698,148.936
C00864=1148.935,119.970,-55.572,-178.988,6.700,148.936
C00865=1148.929,120.219,-55.591,-178.985,6.701,148.935
C00866=1148.925,120.468,-55.611,-178.982,6.703,148.935
C00867=1148.920,120.718,-55.631,-178.980,6.705,148.934
C00868=1148.915,120.966,-55.649,-178.977,6.706,148.934
C00869=1148.910,121.216,-55.669,-178.974,6.708,148.933
C00870=1148.905,121.465,-55.688,-178.971,6.710,148.933
C00871=1148.900,121.714,-55.708,-178.968,6.711,148.933
C00872=1148.896,121.964,-55.728,-178.966,6.713,148.932
C00873=1148.891,122.212,-55.746,-178.963,6.715,148.932
C00874=1148.886,122.462,-55.766,-178.960,6.716,148.931
C00875=1148.881,122.711,-55.785,-178.958,6.718,148.931
C00876=1148.876,122.960,-55.805,-178.955,6.720,148.931
C00877=1148.872,123.209,-55.825,-178.952,6.721,148.930
C00878=1148.866,123.458,-55.845,-178.949,6.723,148.930
C00879=1148.862,123.707,-55.864,-178.947,6.725,148.929
C00880=1148.858,123.957,-55.883,-178.944,6.727,148.929
C00881=1148.852,124.206,-55.903,-178.941,6.728,148.928
C00882=1148.848,124.455,-55.922,-178.938,6.730,148.928
C00883=1148.843,124.705,-55.942,-178.935,6.731,148.928
C00884=1148.838,124.953,-55.962,-178.933,6.733,148.927
C00885=1148.833,125.203,-55.982,-178.930,6.735,148.927
C00886=1148.828,125.452,-56.001,-178.927,6.736,148.926
C00887=1148.824,125.702,-56.020,-178.924,6.738,148.926
C00888=1148.819,125.950,-56.040,-178.922,6.740,148.926
C00889=1148.815,126.199,-56.060,-178.919,6.742,148.925
C00890=1148.810,126.449,-56.080,-178.916,6.743,148.925
C00891=1148.804,126.698,-56.099,-178.914,6.745,148.924
C00892=1148.800,126.947,-56.119,-178.911,6.747,148.924
C00893=1148.795,127.196,-56.139,-178.908,6.748,148.924
C00894=1148.791,127.446,-56.159,-178.905,6.750,148.923
C00895=1148.785,127.694,-56.179,-178.903,6.752,148.923
C00896=1148.781,127.944,-56.198,-178.900,6.753,148.922
C00897=1148.776,128.193,-56.218,-178.897,6.755,148.922
C00898=1148.771,128.442,-56.238,-178.895,6.757,148.922
C00899=1148.766,128.691,-56.258,-178.891,6.758,148.921
C00900=1148.761,128.941,-56.277,-178.889,6.760,148.921
C00901=1148.757,129.190,-56.298,-178.886,6.762,148.920
C00902=1148.752,129.439,-56.317,-178.883,6.763,148.920
C00903=1148.747,129.688,-56.337,-178.880,6.765,148.919
C00904=1148.743,129.937,-56.357,-178.878,6.767,148.919
C00905=1148.738,130.187,-56.377,-178.875,6.768,148.919
C00906=1148.733,130.436,-56.397,-178.872,6.770,148.918
C00907=1148.728,130.684,-56.416,-178.870,6.772,148.918
C00908=1148.724,130.933,-56.437,-178.867,6.774,148.917
C00909=1148.718,131.183,-56.457,-178.864,6.775,148.917
C00910=1148.713,131.451,-56.479,-178.861,6.778,148.917
C00911=1148.709,131.720,-56.500,-178.858,6.780,148.916
C00912=1148.703,131.989,-56.522,-178.855,6.781,148.916
C00913=1148.698,132.257,-56.543,-178.852,6.783,148.915
C00914=1148.694,132.507,-56.563,-178.849,6.785,148.915
C00915=1148.688,132.755,-56.584,-178.846,6.787,148.914
C00916=1148.683,133.005,-56.603,-178.843,6.789,148.914
C00917=1148.679,133.254,-56.624,-178.841,6.790,148.914
C00918=1148.674,133.503,-56.643,-178.838,6.792,148.913
C00919=1148.669,133.752,-56.664,-178.835,6.794,148.913
C00920=1148.665,134.001,-56.684,-178.833,6.795,148.912
C00921=1148.660,134.251,-56.704,-178.830,6.797,148.912
C00922=1148.654,134.499,-56.724,-178.827,6.799,148.912
C00923=1148.650,134.748,-56.745,-178.824,6.801,148.911
C00924=1148.645,134.998,-56.764,-178.822,6.802,148.911
C00925=1148.641,135.247,-56.785,-178.819,6.804,148.910
C00926=1148.636,135.496,-56.805,-178.816,6.806,148.910
C00927=1148.631,135.746,-56.825,-178.813,6.808,148.910
C00928=1148.626,135.994,-56.846,-178.810,6.810,148.909
C00929=1148.622,136.243,-56.866,-178.808,6.812,148.909
C00930=1148.617,136.492,-56.885,-178.805,6.813,148.909
C00931=1148.612,136.742,-56.906,-178.802,6.815,148.908
C00932=1148.607,136.990,-56.927,-178.799,6.817,148.908
C00933=1148.603,137.239,-56.947,-178.797,6.818,148.907
C00934=1148.598,137.489,-56.967,-178.794,6.820,148.907
C00935=1148.593,137.738,-56.988,-178.791,6.822,148.907
C00936=1148.588,137.987,-57.008,-178.788,6.825,148.906
C00937=1148.584,138.236,-57.028,-178.786,6.826,148.906
C00938=1148.578,138.486,-57.049,-178.783,6.828,148.906
C00939=1148.574,138.735,-57.069,-178.780,6.830,148.905
C00940=1148.570,138.984,-57.089,-178.778,6.832,148.905
C00941=1148.564,139.233,-57.110,-178.775,6.833,148.904
C00942=1148.560,139.482,-57.131,-178.772,6.835,148.904
C00943=1148.555,139.731,-57.151,-178.770,6.837,148.904
C00944=1148.550,139.980,-57.172,-178.767,6.838,148.903
C00945=1148.546,140.230,-57.192,-178.763,6.841,148.903
C00946=1148.541,140.479,-57.212,-178.761,6.843,148.903
C00947=1148.536,140.728,-57.233,-178.758,6.844,148.902
C00948=1148.531,140.977,-57.253,-178.755,6.846,148.902
C00949=1148.527,141.226,-57.274,-178.753,6.848,148.901
C00950=1148.522,141.475,-57.295,-178.750,6.850,148.901
C00951=1148.517,141.724,-57.315,-178.747,6.851,148.901
C00952=1148.512,141.973,-57.336,-178.744,6.854,148.900
C00953=1148.508,142.222,-57.357,-178.741,6.855,148.900
C00954=1148.503,142.471,-57.377,-178.739,6.857,148.899
C00955=1148.498,142.721,-57.398,-178.736,6.859,148.899
C00956=1148.494,142.970,-57.418,-178.733,6.861,148.899
C00957=1148.489,143.219,-57.439,-178.730,6.862,148.898
C00958=1148.484,143.468,-57.460,-178.728,6.864,148.898
C00959=1148.479,143.717,-57.481,-178.724,6.867,148.898
C00960=1148.475,143.966,-57.501,-178.722,6.869,148.897
C00961=1148.469,144.215,-57.522,-178.719,6.870,148.897
C00962=1148.465,144.464,-57.542,-178.717,6.872,148.897
C00963=1148.460,144.713,-57.563,-178.714,6.874,148.896
C00964=1148.456,144.962,-57.584,-178.711,6.876,148.896
C00965=1148.450,145.211,-57.605,-178.709,6.877,148.895
C00966=1148.446,145.460,-57.626,-178.705,6.880,148.895
C00967=1148.441,145.710,-57.647,-178.703,6.881,148.895
C00968=1148.437,145.959,-57.667,-178.700,6.883,148.894
C00969=1148.432,146.208,-57.688,-178.697,6.885,148.894
C00970=1148.427,146.457,-57.709,-178.694,6.887,148.894
C00971=1148.423,146.706,-57.730,-178.692,6.888,148.893
C00972=1148.418,146.955,-57.751,-178.688,6.891,148.893
C00973=1148.413,147.204,-57.772,-178.686,6.893,148.893
C00974=1148.408,147.453,-57.793,-178.683,6.895,148.892
C00975=1148.404,147.702,-57.814,-178.681,6.896,148.892
C00976=1148.399,147.952,-57.835,-178.678,6.898,148.891
C00977=1148.395,148.200,-57.855,-178.675,6.901,148.891
C00978=1148.389,148.450,-57.876,-178.672,6.902,148.891
C00979=1148.385,148.698,-57.898,-178.669,6.904,148.890
C00980=1148.380,148.947,-57.918,-178.667,6.906,148.890
C00981=1148.375,149.197,-57.939,-178.664,6.908,148.890
C00982=1148.370,149.446,-57.960,-178.661,6.910,148.889
C00983=1148.366,149.695,-57.982,-178.658,6.912,148.889
C00984=1148.361,149.944,-58.003,-178.656,6.914,148.889
C00985=1148.356,150.193,-58.024,-178.653,6.916,148.888
C00986=1148.352,150.442,-58.045,-178.650,6.917,148.888
C00987=1148.347,150.691,-58.066,-178.647,6.920,148.887
C00988=1148.342,150.940,-58.088,-178.644,6.922,148.887
C00989=1148.338,151.189,-58.108,-178.642,6.923,148.887
C00990=1148.333,151.439,-58.129,-178.639,6.925,148.886
C00991=1148.328,151.687,-58.151,-178.636,6.927,148.886
C00992=1148.323,151.936,-58.172,-178.633,6.929,148.886
C00993=1148.319,152.185,-58.193,-178.631,6.931,148.885
C00994=1148.314,152.435,-58.214,-178.628,6.933,148.885
C00995=1148.309,152.683,-58.236,-178.625,6.935,148.885
C00996=1148.304,152.933,-58.257,-178.623,6.936,148.884
C00997=1148.300,153.181,-58.278,-178.619,6.939,148.884
C00998=1148.295,153.431,-58.299,-178.617,6.941,148.884
C00999=1148.290,153.680,-58.321,-178.614,6.942,148.883
C01000=1148.285,153.929,-58.342,-178.612,6.945,148.883
C01001=1148.280,154.177,-58.364,-178.608,6.947,148.883
C01002=1148.276,154.427,-58.384,-178.606,6.949,148.882
C01003=1148.272,154.676,-58.406,-178.603,6.951,148.882
C01004=1148.266,154.925,-58.427,-178.600,6.952,148.881
C01005=1148.262,155.174,-58.449,-178.597,6.955,148.881
C01006=1148.257,155.424,-58.470,-178.594,6.956,148.881
C01007=1148.253,155.672,-58.491,-178.592,6.959,148.881
C01008=1148.248,155.921,-58.513,-178.589,6.960,148.880
C01009=1148.243,156.171,-58.534,-178.586,6.963,148.880
C01010=1148.239,156.419,-58.556,-178.583,6.965,148.879
C01011=1148.234,156.668,-58.578,-178.581,6.966,148.879
C01012=1148.229,156.918,-58.599,-178.578,6.968,148.879
C01013=1148.224,157.166,-58.621,-178.575,6.971,148.878
C01014=1148.219,157.435,-58.643,-178.572,6.972,148.878
C01015=1148.214,157.704,-58.667,-178.569,6.975,148.878
C01016=1148.210,157.973,-58.690,-178.566,6.977,148.877
C01017=1148.204,158.243,-58.714,-178.563,6.979,148.877
C01018=1148.199,158.491,-58.735,-178.560,6.981,148.877
C01019=1148.194,158.740,-58.757,-178.558,6.983,148.876
C01020=1148.190,158.990,-58.778,-178.555,6.985,148.876
C01021=1148.185,159.239,-58.800,-178.552,6.987,148.876
C01022=1148.180,159.487,-58.822,-178.549,6.989,148.875
C01023=1148.176,159.736,-58.843,-178.547,6.991,148.875
C01024=1148.172,159.985,-58.865,-178.544,6.993,148.875
C01025=1148.166,160.234,-58.886,-178.541,6.995,148.874
C01026=1148.162,160.483,-58.908,-178.538,6.997,148.874
C01027=1148.157,160.732,-58.929,-178.535,6.999,148.874
C01028=1148.153,160.981,-58.951,-178.532,7.002,148.873
C01029=1148.148,161.230,-58.973,-178.530,7.003,148.873
C01030=1148.143,161.479,-58.995,-178.527,7.005,148.873
C01031=1148.138,161.728,-59.018,-178.524,7.007,148.872
C01032=1148.133,161.977,-59.039,-178.521,7.009,148.872
C01033=1148.129,162.227,-59.061,-178.519,7.011,148.872
C01034=1148.124,162.476,-59.082,-178.516,7.013,148.871
C01035=1148.120,162.725,-59.104,-178.513,7.016,148.871
C01036=1148.115,162.974,-59.126,-178.510,7.017,148.871
C01037=1148.110,163.222,-59.148,-178.507,7.019,148.870
C01038=1148.106,163.472,-59.170,-178.505,7.022,148.870
C01039=1148.101,163.720,-59.191,-178.502,7.024,148.870
C01040=1148.097,163.970,-59.213,-178.499,7.025,148.869
C01041=1148.092,164.218,-59.235,-178.497,7.027,148.869
C01042=1148.087,164.467,-59.257,-178.493,7.030,148.869
C01043=1148.083,164.716,-59.279,-178.491,7.032,148.869
C01044=1148.078,164.966,-59.301,-178.488,7.033,148.868
C01045=1148.073,165.214,-59.323,-178.485,7.036,148.868
C01046=1148.068,165.464,-59.345,-178.482,7.038,148.867
C01047=1148.064,165.712,-59.368,-178.480,7.040,148.867
C01048=1148.060,165.961,-59.390,-178.477,7.042,148.867
C01049=1148.055,166.210,-59.411,-178.474,7.044,148.867
C01050=1148.050,166.459,-59.434,-178.471,7.046,148.866
C01051=1148.045,166.708,-59.456,-178.468,7.048,148.866
C01052=1148.041,166.957,-59.478,-178.466,7.050,148.866
C01053=1148.036,167.206,-59.499,-178.463,7.052,148.865
C01054=1148.031,167.455,-59.521,-178.460,7.055,148.865
C01055=1148.026,167.704,-59.544,-178.457,7.056,148.865
C01056=1148.022,167.953,-59.566,-178.455,7.059,148.864
C01057=1148.017,168.202,-59.588,-178.452,7.061,148.864
C01058=1148.013,168.451,-59.610,-178.449,7.063,148.864
C01059=1148.007,168.700,-59.632,-178.446,7.065,148.863
C01060=1148.003,168.949,-59.655,-178.443,7.067,148.863
C01061=1147.999,169.198,-59.677,-178.441,7.069,148.863
C01062=1147.993,169.447,-59.700,-178.438,7.071,148.862
C01063=1147.989,169.696,-59.722,-178.435,7.073,148.862
C01064=1147.984,169.944,-59.744,-178.433,7.076,148.862
C01065=1147.980,170.194,-59.766,-178.430,7.077,148.862
C01066=1147.975,170.443,-59.788,-178.427,7.080,148.861
C01067=1147.971,170.691,-59.811,-178.424,7.082,148.861
C01068=1147.966,170.941,-59.833,-178.421,7.084,148.861
C01069=1147.961,171.190,-59.855,-178.418,7.086,148.860
C01070=1147.957,171.438,-59.878,-178.416,7.088,148.860
C01071=1147.951,171.687,-59.900,-178.413,7.091,148.860
C01072=1147.947,171.937,-59.923,-178.410,7.093,148.860
C01073=1147.943,172.185,-59.945,-178.407,7.094,148.859
C01074=1147.937,172.434,-59.968,-178.404,7.097,148.859
C01075=1147.933,172.683,-59.990,-178.402,7.099,148.859
C01076=1147.929,172.932,-60.012,-178.399,7.101,148.858
C01077=1147.923,173.181,-60.035,-178.396,7.103,148.858
C01078=1147.920,173.430,-60.057,-178.394,7.105,148.858
C01079=1147.915,173.680,-60.080,-178.390,7.108,148.857
C01080=1147.910,173.928,-60.102,-178.388,7.110,148.857
C01081=1147.905,174.177,-60.125,-178.386,7.112,148.857
C01082=1147.901,174.426,-60.148,-178.382,7.114,148.857
C01083=1147.896,174.675,-60.170,-178.380,7.116,148.856
C01084=1147.891,174.924,-60.193,-178.376,7.118,148.856
C01085=1147.887,175.173,-60.215,-178.374,7.121,148.856
C01086=1147.882,175.421,-60.238,-178.371,7.122,148.855
C01087=1147.878,175.670,-60.261,-178.368,7.125,148.855
C01088=1147.873,175.920,-60.283,-178.366,7.127,148.855
C01089=1147.868,176.168,-60.306,-178.363,7.129,148.855
C01090=1147.863,176.418,-60.328,-178.360,7.131,148.854
C01091=1147.859,176.666,-60.351,-178.358,7.133,148.854
C01092=1147.855,176.915,-60.375,-178.354,7.136,148.854
C01093=1147.850,177.164,-60.396,-178.352,7.138,148.853
C01094=1147.845,177.413,-60.420,-178.349,7.140,148.853
C01095=1147.841,177.662,-60.442,-178.346,7.142,148.853
C01096=1147.836,177.911,-60.465,-178.344,7.144,148.852
C01097=1147.831,178.160,-60.488,-178.341,7.147,148.852
C01098=1147.827,178.408,-60.511,-178.338,7.149,148.852
C01099=1147.822,178.658,-60.533,-178.335,7.151,148.852
C01100=1147.818,178.907,-60.556,-178.332,7.153,148.851
C01101=1147.813,179.155,-60.579,-178.329,7.156,148.851
C01102=1147.808,179.405,-60.602,-178.327,7.158,148.851
C01103=1147.804,179.653,-60.625,-178.324,7.160,148.851
C01104=1147.799,179.902,-60.648,-178.321,7.162,148.850
C01105=1147.794,180.150,-60.670,-178.318,7.164,148.850
C01106=1147.790,180.400,-60.694,-178.316,7.167,148.850
C01107=1147.785,180.649,-60.716,-178.313,7.169,148.849
C01108=1147.781,180.898,-60.739,-178.310,7.171,148.849
C01109=1147.776,181.147,-60.762,-178.307,7.173,148.849
C01110=1147.771,181.396,-60.786,-178.305,7.175,148.849
C01111=1147.767,181.644,-60.808,-178.301,7.177,148.848
C01112=1147.762,181.893,-60.832,-178.299,7.180,148.848
C01113=1147.757,182.143,-60.854,-178.296,7.182,148.848
C01114=1147.753,182.391,-60.877,-178.294,7.184,148.848
C01115=1147.748,182.640,-60.900,-178.290,7.187,148.847
C01116=1147.744,182.889,-60.924,-178.288,7.188,148.847
C01117=1147.738,183.138,-60.947,-178.285,7.191,148.847
C01118=1147.734,183.408,-60.971,-178.282,7.193,148.846
C01119=1147.729,183.678,-60.996,-178.279,7.196,148.846
C01120=1147.724,183.947,-61.022,-178.276,7.198,148.846
C01121=1147.719,184.216,-61.047,-178.273,7.201,148.846
C01122=1147.715,184.465,-61.070,-178.270,7.203,148.845
C01123=1147.710,184.714,-61.093,-178.267,7.205,148.845
C01124=1147.705,184.963,-61.117,-178.265,7.208,148.845
C01125=1147.700,185.212,-61.140,-178.262,7.209,148.844
C01126=1147.696,185.460,-61.162,-178.259,7.212,148.844
C01127=1147.691,185.709,-61.186,-178.256,7.214,148.844
C01128=1147.687,185.959,-61.209,-178.253,7.216,148.844
C01129=1147.682,186.208,-61.233,-178.251,7.219,148.843
C01130=1147.677,186.457,-61.256,-178.248,7.221,148.843
C01131=1147.673,186.706,-61.279,-178.245,7.223,148.843
C01132=1147.669,186.954,-61.303,-178.242,7.226,148.843
C01133=1147.664,187.203,-61.326,-178.240,7.228,148.843
C01134=1147.660,187.452,-61.349,-178.237,7.230,148.842
C01135=1147.655,187.701,-61.373,-178.234,7.232,148.842
C01136=1147.650,187.950,-61.396,-178.231,7.235,148.842
C01137=1147.645,188.199,-61.420,-178.228,7.237,148.841
C01138=1147.641,188.448,-61.443,-178.226,7.240,148.841
C01139=1147.636,188.696,-61.467,-178.223,7.241,148.841
C01140=1147.631,188.945,-61.490,-178.220,7.244,148.841
C01141=1147.626,189.194,-61.513,-178.217,7.246,148.840
C01142=1147.622,189.442,-61.536,-178.214,7.249,148.840
C01143=1147.618,189.691,-61.560,-178.212,7.251,148.840
C01144=1147.613,189.940,-61.584,-178.209,7.253,148.840
C01145=1147.609,190.189,-61.607,-178.206,7.255,148.839
C01146=1147.604,190.438,-61.630,-178.203,7.258,148.839
C01147=1147.600,190.686,-61.654,-178.201,7.260,148.839
C01148=1147.595,190.935,-61.678,-178.198,7.263,148.839
C01149=1147.590,191.184,-61.701,-178.195,7.264,148.838
C01150=1147.586,191.433,-61.725,-178.192,7.267,148.838
C01151=1147.581,191.682,-61.748,-178.190,7.269,148.838
C01152=1147.576,191.931,-61.772,-178.187,7.272,148.838
C01153=1147.572,192.179,-61.796,-178.184,7.274,148.837
C01154=1147.568,192.429,-61.820,-178.181,7.277,148.837
C01155=1147.563,192.677,-61.844,-178.178,7.279,148.837
C01156=1147.558,192.927,-61.868,-178.176,7.281,148.837
C01157=1147.553,193.176,-61.891,-178.172,7.284,148.836
C01158=1147.549,193.424,-61.915,-178.170,7.286,148.836
C01159=1147.544,193.673,-61.938,-178.167,7.288,148.836
C01160=1147.540,193.922,-61.963,-178.165,7.290,148.836
C01161=1147.535,194.171,-61.986,-178.161,7.293,148.835
C01162=1147.531,194.419,-62.010,-178.159,7.295,148.835
C01163=1147.526,194.668,-62.033,-178.156,7.298,148.835
C01164=1147.522,194.917,-62.057,-178.153,7.299,148.835
C01165=1147.517,195.166,-62.081,-178.150,7.302,148.835
C01166=1147.512,195.414,-62.105,-178.147,7.305,148.834
C01167=1147.508,195.664,-62.129,-178.145,7.307,148.834
C01168=1147.503,195.912,-62.153,-178.142,7.310,148.834
C01169=1147.499,196.162,-62.177,-178.140,7.312,148.834
C01170=1147.494,196.410,-62.201,-178.136,7.314,148.833
C01171=1147.490,196.658,-62.225,-178.134,7.316,148.833
C01172=1147.484,196.908,-62.249,-178.131,7.319,148.833
C01173=1147.480,197.156,-62.273,-178.129,7.321,148.833
C01174=1147.476,197.405,-62.297,-178.125,7.324,148.832
C01175=1147.471,197.654,-62.321,-178.122,7.326,148.832
C01176=1147.467,197.903,-62.345,-178.120,7.328,148.832
C01177=1147.462,198.151,-62.369,-178.117,7.331,148.832
C01178=1147.457,198.400,-62.393,-178.115,7.333,148.832
C01179=1147.453,198.649,-62.417,-178.111,7.336,148.831
C01180=1147.449,198.898,-62.441,-178.109,7.338,148.831
C01181=1147.444,199.147,-62.465,-178.106,7.340,148.831
C01182=1147.439,199.396,-62.489,-178.103,7.343,148.831
C01183=1147.435,199.644,-62.513,-178.101,7.345,148.830
C01184=1147.430,199.892,-62.537,-178.098,7.348,148.830
C01185=1147.426,200.143,-62.562,-178.095,7.350,148.830
C01186=1147.421,200.391,-62.586,-178.092,7.353,148.830
C01187=1147.417,200.639,-62.610,-178.089,7.355,148.830
C01188=1147.412,200.888,-62.635,-178.087,7.357,148.829
C01189=1147.407,201.137,-62.659,-178.083,7.360,148.829
C01190=1147.403,201.386,-62.682,-178.081,7.362,148.829
C01191=1147.398,201.635,-62.707,-178.078,7.365,148.829
C01192=1147.394,201.883,-62.731,-178.075,7.367,148.829
C01193=1147.389,202.132,-62.755,-178.073,7.370,148.828
C01194=1147.385,202.381,-62.780,-178.070,7.372,148.828
C01195=1147.380,202.630,-62.804,-178.067,7.374,148.828
C01196=1147.376,202.878,-62.828,-178.064,7.377,148.828
C01197=1147.371,203.127,-62.853,-178.061,7.380,148.827
C01198=1147.367,203.376,-62.877,-178.059,7.381,148.827
C01199=1147.362,203.625,-62.902,-178.056,7.384,148.827
C01200=1147.358,203.873,-62.926,-178.053,7.386,148.827
C01201=1147.354,204.122,-62.951,-178.050,7.389,148.827
C01202=1147.349,204.371,-62.975,-178.048,7.392,148.826
C01203=1147.344,204.619,-62.999,-178.045,7.394,148.826
C01204=1147.340,204.869,-63.024,-178.042,7.397,148.826
C01205=1147.335,205.117,-63.048,-178.039,7.399,148.826
C01206=1147.330,205.366,-63.073,-178.037,7.401,148.826
C01207=1147.326,205.615,-63.098,-178.034,7.404,148.825
C01208=1147.321,205.864,-63.122,-178.031,7.406,148.825
C01209=1147.317,206.112,-63.146,-178.028,7.409,148.825
C01210=1147.312,206.361,-63.171,-178.025,7.411,148.825
C01211=1147.308,206.610,-63.195,-178.023,7.413,148.825
C01212=1147.303,206.859,-63.220,-178.020,7.416,148.824
C01213=1147.299,207.108,-63.245,-178.017,7.419,148.824
C01214=1147.294,207.356,-63.269,-178.015,7.421,148.824
C01215=1147.290,207.604,-63.294,-178.011,7.424,148.824
C01216=1147.285,207.854,-63.319,-178.009,7.427,148.824
C01217=1147.281,208.102,-63.343,-178.006,7.429,148.823
C01218=1147.276,208.351,-63.368,-178.003,7.431,148.823
C01219=1147.271,208.600,-63.393,-178.000,7.434,148.823
C01220=1147.267,208.849,-63.417,-177.998,7.436,148.823
C01221=1147.263,209.097,-63.443,-177.995,7.439,148.823
C01222=1147.257,209.368,-63.469,-177.992,7.442,148.823
C01223=1147.253,209.639,-63.496,-177.989,7.444,148.822
C01224=1147.248,209.909,-63.523,-177.986,7.447,148.822
C01225=1147.243,210.180,-63.550,-177.983,7.450,148.822
C01226=1147.238,210.428,-63.575,-177.980,7.452,148.822
C01227=1147.233,210.677,-63.600,-177.977,7.454,148.821
C01228=1147.229,210.925,-63.625,-177.974,7.457,148.821
C01229=1147.224,211.174,-63.649,-177.972,7.459,148.821
C01230=1147.220,211.424,-63.674,-177.969,7.462,148.821
C01231=1147.216,211.671,-63.699,-177.966,7.465,148.821
C01232=1147.211,211.921,-63.724,-177.964,7.467,148.821
C01233=1147.206,212.170,-63.749,-177.961,7.470,148.820
C01234=1147.202,212.418,-63.774,-177.958,7.472,148.820
C01235=1147.197,212.667,-63.799,-177.955,7.475,148.820
C01236=1147.193,212.916,-63.824,-177.952,7.477,148.820
C01237=1147.188,213.164,-63.849,-177.950,7.480,148.820
C01238=1147.185,213.413,-63.874,-177.947,7.483,148.820
C01239=1147.179,213.662,-63.899,-177.944,7.485,148.819
C01240=1147.175,213.910,-63.925,-177.941,7.488,148.819
C01241=1147.170,214.159,-63.949,-177.938,7.491,148.819
C01242=1147.167,214.408,-63.975,-177.936,7.492,148.819
C01243=1147.161,214.656,-63.999,-177.933,7.495,148.819
C01244=1147.157,214.905,-64.025,-177.930,7.498,148.818
C01245=1147.152,215.154,-64.050,-177.927,7.501,148.818
C01246=1147.149,215.402,-64.075,-177.925,7.503,148.818
C01247=1147.143,215.651,-64.099,-177.922,7.506,148.818
C01248=1147.139,215.900,-64.125,-177.919,7.508,148.818
C01249=1147.134,216.149,-64.150,-177.916,7.510,148.817
C01250=1147.130,216.397,-64.176,-177.914,7.513,148.817
C01251=1147.125,216.645,-64.201,-177.910,7.516,148.817
C01252=1147.120,216.895,-64.226,-177.908,7.519,148.817
C01253=1147.117,217.143,-64.251,-177.905,7.521,148.817
C01254=1147.112,217.391,-64.277,-177.903,7.524,148.817
C01255=1147.108,217.641,-64.302,-177.899,7.526,148.816
C01256=1147.103,217.889,-64.327,-177.897,7.528,148.816
C01257=1147.099,218.138,-64.353,-177.894,7.531,148.816
C01258=1147.094,218.387,-64.378,-177.891,7.534,148.816
C01259=1147.089,218.635,-64.403,-177.888,7.537,148.816
C01260=1147.085,218.884,-64.429,-177.886,7.539,148.816
C01261=1147.080,219.132,-64.454,-177.883,7.542,148.816
C01262=1147.076,219.382,-64.479,-177.880,7.544,148.815
C01263=1147.072,219.630,-64.505,-177.877,7.547,148.815
C01264=1147.067,219.878,-64.530,-177.875,7.549,148.815
C01265=1147.063,220.127,-64.556,-177.872,7.552,148.815
C01266=1147.059,220.376,-64.581,-177.869,7.555,148.815
C01267=1147.054,220.625,-64.606,-177.866,7.558,148.815
C01268=1147.050,220.873,-64.632,-177.864,7.560,148.814
C01269=1147.045,221.122,-64.657,-177.861,7.563,148.814
C01270=1147.040,221.370,-64.683,-177.858,7.566,148.814
C01271=1147.036,221.619,-64.709,-177.855,7.568,148.814
C01272=1147.031,221.867,-64.734,-177.853,7.571,148.814
C01273=1147.027,222.116,-64.760,-177.850,7.573,148.814
C01274=1147.022,222.365,-64.786,-177.847,7.576,148.813
C01275=1147.017,222.614,-64.811,-177.844,7.579,148.813
C01276=1147.013,222.863,-64.837,-177.842,7.581,148.813
C01277=1147.009,223.112,-64.862,-177.839,7.584,148.813
C01278=1147.004,223.360,-64.888,-177.836,7.587,148.813
C01279=1147.000,223.608,-64.913,-177.833,7.589,148.813
C01280=1146.995,223.857,-64.939,-177.831,7.592,148.813
C01281=1146.991,224.106,-64.965,-177.828,7.594,148.812
C01282=1146.986,224.354,-64.990,-177.825,7.597,148.812
C01283=1146.982,224.603,-65.016,-177.822,7.600,148.812
C01284=1146.978,224.852,-65.042,-177.819,7.603,148.812
C01285=1146.973,225.101,-65.068,-177.817,7.605,148.812
C01286=1146.968,225.348,-65.094,-177.814,7.608,148.812
C01287=1146.964,225.597,-65.120,-177.811,7.610,148.812
C01288=1146.960,225.846,-65.146,-177.808,7.613,148.811
C01289=1146.956,226.095,-65.172,-177.805,7.616,148.811
C01290=1146.951,226.343,-65.197,-177.803,7.618,148.811
C01291=1146.946,226.592,-65.223,-177.800,7.621,148.811
C01292=1146.942,226.841,-65.249,-177.797,7.624,148.811
C01293=1146.937,227.090,-65.275,-177.794,7.627,148.811
C01294=1146.934,227.338,-65.301,-177.791,7.630,148.811
C01295=1146.928,227.586,-65.327,-177.789,7.632,148.811
C01296=1146.924,227.835,-65.353,-177.786,7.634,148.810
C01297=1146.920,228.084,-65.379,-177.783,7.637,148.810
C01298=1146.915,228.333,-65.405,-177.780,7.640,148.810
C01299=1146.911,228.581,-65.432,-177.778,7.643,148.810
C01300=1146.906,228.829,-65.457,-177.775,7.645,148.810
C01301=1146.902,229.078,-65.483,-177.772,7.648,148.810
C01302=1146.898,229.326,-65.509,-177.769,7.651,148.809
C01303=1146.893,229.575,-65.536,-177.767,7.654,148.809
C01304=1146.889,229.824,-65.561,-177.764,7.657,148.809
C01305=1146.884,230.073,-65.587,-177.761,7.660,148.809
C01306=1146.879,230.321,-65.614,-177.758,7.661,148.809
C01307=1146.875,230.569,-65.639,-177.756,7.664,148.809
C01308=1146.871,230.818,-65.666,-177.753,7.667,148.809
C01309=1146.866,231.067,-65.692,-177.750,7.670,148.809
C01310=1146.862,231.316,-65.718,-177.747,7.673,148.809
C01311=1146.858,231.564,-65.745,-177.745,7.675,148.808
C01312=1146.853,231.813,-65.771,-177.742,7.678,148.808
C01313=1146.849,232.061,-65.797,-177.739,7.681,148.808
C01314=1146.843,232.309,-65.823,-177.736,7.684,148.808
C01315=1146.839,232.558,-65.849,-177.733,7.686,148.808
C01316=1146.835,232.806,-65.876,-177.730,7.689,148.808
C01317=1146.830,233.056,-65.902,-177.728,7.692,148.808
C01318=1146.826,233.304,-65.928,-177.725,7.694,148.808
C01319=1146.821,233.553,-65.955,-177.722,7.697,148.807
C01320=1146.817,233.801,-65.981,-177.719,7.700,148.807
C01321=1146.812,234.050,-66.007,-177.717,7.703,148.807
C01322=1146.809,234.298,-66.034,-177.714,7.706,148.807
C01323=1146.805,234.547,-66.060,-177.711,7.709,148.807
C01324=1146.800,234.796,-66.087,-177.709,7.711,148.807
C01325=1146.796,235.044,-66.113,-177.706,7.714,148.807
C01326=1146.790,235.316,-66.142,-177.702,7.717,148.807
C01327=1146.785,235.588,-66.171,-177.699,7.720,148.806
C01328=1146.781,235.859,-66.200,-177.697,7.723,148.806
C01329=1146.775,236.131,-66.229,-177.694,7.726,148.806
C01330=1146.771,236.380,-66.256,-177.691,7.729,148.806
C01331=1146.767,236.628,-66.282,-177.688,7.732,148.806
C01332=1146.762,236.877,-66.308,-177.685,7.734,148.806
C01333=1146.758,237.125,-66.335,-177.682,7.737,148.806
C01334=1146.753,237.374,-66.362,-177.679,7.740,148.806
C01335=1146.749,237.622,-66.388,-177.677,7.742,148.806
C01336=1146.744,237.871,-66.415,-177.674,7.745,148.805
C01337=1146.740,238.119,-66.442,-177.672,7.748,148.805
C01338=1146.736,238.368,-66.468,-177.669,7.751,148.805
C01339=1146.732,238.617,-66.496,-177.666,7.754,148.805
C01340=1146.728,238.866,-66.522,-177.663,7.757,148.805
C01341=1146.723,239.114,-66.549,-177.661,7.760,148.805
C01342=1146.718,239.363,-66.576,-177.657,7.762,148.805
C01343=1146.714,239.611,-66.602,-177.654,7.765,148.805
C01344=1146.710,239.859,-66.629,-177.652,7.767,148.805
C01345=1146.705,240.108,-66.656,-177.649,7.770,148.805
C01346=1146.701,240.357,-66.682,-177.647,7.773,148.804
C01347=1146.696,240.605,-66.709,-177.644,7.776,148.804
C01348=1146.691,240.854,-66.736,-177.641,7.779,148.804
C01349=1146.688,241.102,-66.763,-177.638,7.782,148.804
C01350=1146.683,241.350,-66.790,-177.636,7.785,148.804
C01351=1146.678,241.599,-66.817,-177.633,7.788,148.804
C01352=1146.674,241.847,-66.844,-177.630,7.791,148.804
C01353=1146.670,242.096,-66.871,-177.627,7.794,148.804
C01354=1146.666,242.345,-66.898,-177.625,7.796,148.804
C01355=1146.661,242.593,-66.925,-177.622,7.799,148.804
C01356=1146.656,242.842,-66.952,-177.619,7.801,148.803
C01357=1146.652,243.090,-66.978,-177.616,7.804,148.803
C01358=1146.648,243.338,-67.005,-177.613,7.807,148.803
C01359=1146.643,243.587,-67.032,-177.611,7.810,148.803
C01360=1146.638,243.835,-67.059,-177.608,7.813,148.803
C01361=1146.635,244.084,-67.086,-177.605,7.816,148.803
C01362=1146.630,244.333,-67.113,-177.602,7.819,148.803
C01363=1146.626,244.581,-67.140,-177.599,7.822,148.803
C01364=1146.621,244.830,-67.167,-177.597,7.825,148.803
C01365=1146.617,245.078,-67.195,-177.594,7.828,148.803
C01366=1146.612,245.326,-67.222,-177.591,7.831,148.803
C01367=1146.609,245.575,-67.249,-177.589,7.833,148.803
C01368=1146.604,245.823,-67.276,-177.586,7.836,148.803
C01369=1146.599,246.072,-67.303,-177.583,7.839,148.802
C01370=1146.595,246.320,-67.330,-177.580,7.841,148.802
C01371=1146.590,246.568,-67.358,-177.578,7.844,148.802
C01372=1146.586,246.818,-67.386,-177.575,7.847,148.802
C01373=1146.582,247.066,-67.413,-177.572,7.850,148.802
C01374=1146.577,247.315,-67.440,-177.569,7.853,148.802
C01375=1146.573,247.562,-67.467,-177.567,7.856,148.802
C01376=1146.568,247.811,-67.494,-177.564,7.859,148.802
C01377=1146.564,248.060,-67.522,-177.561,7.862,148.802
C01378=1146.560,248.308,-67.548,-177.558,7.865,148.802
C01379=1146.556,248.556,-67.576,-177.555,7.868,148.802
C01380=1146.551,248.805,-67.603,-177.553,7.871,148.802
C01381=1146.547,249.054,-67.631,-177.550,7.874,148.802
C01382=1146.543,249.302,-67.658,-177.547,7.877,148.801
C01383=1146.538,249.550,-67.685,-177.544,7.880,148.801
C01384=1146.534,249.799,-67.714,-177.541,7.882,148.801
C01385=1146.530,250.047,-67.741,-177.539,7.885,148.801
C01386=1146.525,250.296,-67.768,-177.536,7.887,148.801
C01387=1146.521,250.544,-67.796,-177.534,7.890,148.801
C01388=1146.517,250.793,-67.823,-177.531,7.893,148.801
C01389=1146.511,251.041,-67.851,-177.528,7.896,148.801
C01390=1146.507,251.290,-67.878,-177.525,7.899,148.801
C01391=1146.503,251.538,-67.907,-177.523,7.902,148.801
C01392=1146.498,251.787,-67.934,-177.520,7.905,148.801
C01393=1146.494,252.034,-67.961,-177.517,7.908,148.801
C01394=1146.490,252.284,-67.989,-177.514,7.911,148.801
C01395=1146.486,252.532,-68.017,-177.511,7.914,148.801
C01396=1146.481,252.780,-68.044,-177.509,7.917,148.800
C01397=1146.477,253.029,-68.072,-177.506,7.920,148.800
C01398=1146.473,253.277,-68.099,-177.503,7.923,148.801
C01399=1146.468,253.525,-68.127,-177.501,7.926,148.800
C01400=1146.464,253.774,-68.155,-177.498,7.929,148.800
C01401=1146.459,254.022,-68.182,-177.495,7.932,148.800
C01402=1146.455,254.270,-68.210,-177.492,7.935,148.800
C01403=1146.451,254.519,-68.238,-177.490,7.938,148.800
C01404=1146.446,254.767,-68.265,-177.487,7.941,148.800
C01405=1146.443,255.016,-68.294,-177.484,7.943,148.800
C01406=1146.437,255.265,-68.321,-177.481,7.946,148.800
C01407=1146.433,255.513,-68.349,-177.478,7.949,148.800
C01408=1146.429,255.761,-68.377,-177.476,7.952,148.800
C01409=1146.425,256.009,-68.405,-177.473,7.955,148.800
C01410=1146.420,256.259,-68.433,-177.470,7.958,148.800
C01411=1146.416,256.506,-68.461,-177.467,7.961,148.800
C01412=1146.411,256.754,-68.488,-177.465,7.964,148.800
C01413=1146.407,257.003,-68.517,-177.462,7.967,148.800
C01414=1146.402,257.252,-68.544,-177.459,7.970,148.800
C01415=1146.398,257.500,-68.572,-177.457,7.973,148.800
C01416=1146.394,257.748,-68.600,-177.454,7.976,148.800
C01417=1146.390,257.997,-68.628,-177.451,7.979,148.800
C01418=1146.385,258.245,-68.657,-177.448,7.982,148.799
C01419=1146.381,258.493,-68.685,-177.445,7.985,148.799
C01420=1146.377,258.742,-68.712,-177.443,7.988,148.799
C01421=1146.372,258.991,-68.741,-177.440,7.991,148.799
C01422=1146.368,259.239,-68.768,-177.438,7.994,148.799
C01423=1146.364,259.487,-68.796,-177.435,7.997,148.799
C01424=1146.359,259.735,-68.825,-177.432,8.000,148.799
C01425=1146.355,259.983,-68.853,-177.429,8.003,148.799
C01426=1146.350,260.232,-68.881,-177.426,8.006,148.799
C01427=1146.346,260.480,-68.909,-177.424,8.009,148.799
C01428=1146.342,260.729,-68.937,-177.421,8.011,148.799
C01429=1146.338,260.978,-68.966,-177.418,8.014,148.799
C01430=1146.333,261.251,-68.997,-177.415,8.018,148.799
C01431=1146.328,261.524,-69.027,-177.412,8.021,148.799
C01432=1146.323,261.798,-69.059,-177.409,8.025,148.799
C01433=1146.319,262.071,-69.090,-177.406,8.028,148.799
C01434=1146.314,262.320,-69.119,-177.403,8.031,148.799
C01435=1146.310,262.567,-69.147,-177.401,8.034,148.799
C01436=1146.305,262.816,-69.175,-177.398,8.037,148.799
C01437=1146.301,263.064,-69.203,-177.395,8.040,148.799
C01438=1146.297,263.313,-69.231,-177.392,8.043,148.799
C01439=1146.293,263.562,-69.260,-177.390,8.046,148.799
C01440=1146.288,263.810,-69.288,-177.387,8.050,148.799
C01441=1146.284,264.058,-69.317,-177.384,8.053,148.799
C01442=1146.279,264.306,-69.346,-177.381,8.056,148.799
C01443=1146.275,264.555,-69.374,-177.378,8.059,148.799
C01444=1146.271,264.803,-69.403,-177.375,8.061,148.799
C01445=1146.266,265.051,-69.430,-177.373,8.065,148.799
C01446=1146.262,265.300,-69.460,-177.370,8.068,148.799
C01447=1146.258,265.547,-69.488,-177.368,8.071,148.799
C01448=1146.253,265.796,-69.516,-177.365,8.074,148.799
C01449=1146.249,266.045,-69.545,-177.362,8.076,148.799
C01450=1146.245,266.292,-69.573,-177.360,8.080,148.799
C01451=1146.240,266.541,-69.602,-177.357,8.083,148.799
C01452=1146.236,266.789,-69.630,-177.354,8.086,148.799
C01453=1146.232,267.037,-69.659,-177.351,8.089,148.798
C01454=1146.227,267.286,-69.688,-177.349,8.091,148.798
C01455=1146.223,267.534,-69.716,-177.346,8.095,148.799
C01456=1146.219,267.783,-69.745,-177.343,8.098,148.799
C01457=1146.214,268.031,-69.774,-177.340,8.101,148.799
C01458=1146.210,268.279,-69.802,-177.337,8.104,148.798
C01459=1146.206,268.528,-69.831,-177.335,8.107,148.798
C01460=1146.201,268.776,-69.860,-177.332,8.111,148.799
C01461=1146.198,269.024,-69.889,-177.329,8.113,148.798
C01462=1146.193,269.273,-69.917,-177.327,8.116,148.798
C01463=1146.189,269.521,-69.947,-177.324,8.119,148.798
C01464=1146.185,269.769,-69.975,-177.322,8.123,148.799
C01465=1146.180,270.017,-70.004,-177.319,8.126,148.798
C01466=1146.176,270.266,-70.033,-177.316,8.128,148.798
C01467=1146.171,270.514,-70.062,-177.313,8.132,148.798
C01468=1146.168,270.763,-70.090,-177.310,8.135,148.799
C01469=1146.163,271.010,-70.119,-177.307,8.138,148.798
C01470=1146.158,271.259,-70.148,-177.305,8.141,148.798
C01471=1146.154,271.507,-70.178,-177.302,8.144,148.798
C01472=1146.150,271.756,-70.206,-177.300,8.148,148.799
C01473=1146.146,272.004,-70.235,-177.297,8.150,148.798
C01474=1146.142,272.252,-70.264,-177.294,8.153,148.798
C01475=1146.137,272.501,-70.293,-177.291,8.156,148.798
C01476=1146.133,272.749,-70.323,-177.289,8.160,148.799
C01477=1146.128,272.997,-70.352,-177.286,8.163,148.799
C01478=1146.124,273.245,-70.380,-177.283,8.166,148.798
C01479=1146.120,273.493,-70.409,-177.280,8.169,148.798
C01480=1146.116,273.742,-70.439,-177.278,8.172,148.799
C01481=1146.111,273.991,-70.467,-177.275,8.175,148.799
C01482=1146.107,274.238,-70.496,-177.272,8.178,148.798
C01483=1146.102,274.486,-70.526,-177.270,8.182,148.799
C01484=1146.098,274.735,-70.555,-177.267,8.185,148.799
C01485=1146.095,274.983,-70.584,-177.264,8.187,148.799
C01486=1146.090,275.232,-70.613,-177.261,8.192,148.799
C01487=1146.086,275.480,-70.642,-177.259,8.195,148.799
C01488=1146.081,275.727,-70.672,-177.256,8.197,148.799
C01489=1146.077,275.976,-70.701,-177.253,8.200,148.799
C01490=1146.073,276.224,-70.730,-177.251,8.204,148.799
C01491=1146.069,276.473,-70.759,-177.248,8.207,148.799
C01492=1146.064,276.721,-70.789,-177.245,8.210,148.799
C01493=1146.060,276.969,-70.818,-177.243,8.213,148.799
C01494=1146.056,277.218,-70.848,-177.239,8.217,148.799
C01495=1146.051,277.465,-70.877,-177.237,8.219,148.799
C01496=1146.047,277.713,-70.906,-177.234,8.223,148.799
C01497=1146.043,277.962,-70.936,-177.231,8.226,148.799
C01498=1146.039,278.210,-70.965,-177.229,8.229,148.799
C01499=1146.035,278.458,-70.994,-177.226,8.232,148.799
C01500=1146.030,278.706,-71.024,-177.224,8.235,148.799
C01501=1146.026,278.955,-71.053,-177.220,8.239,148.799
C01502=1146.022,279.203,-71.083,-177.218,8.242,148.799
C01503=1146.018,279.451,-71.112,-177.215,8.245,148.799
C01504=1146.014,279.700,-71.142,-177.212,8.248,148.799
C01505=1146.009,279.948,-71.171,-177.210,8.251,148.799
C01506=1146.005,280.196,-71.201,-177.207,8.254,148.799
C01507=1146.001,280.444,-71.230,-177.204,8.258,148.799
C01508=1145.996,280.693,-71.260,-177.202,8.261,148.799
C01509=1145.991,280.940,-71.289,-177.199,8.264,148.799
C01510=1145.987,281.189,-71.319,-177.196,8.267,148.799
C01511=1145.983,281.437,-71.348,-177.194,8.270,148.799
C01512=1145.979,281.685,-71.378,-177.191,8.273,148.799
C01513=1145.975,281.933,-71.408,-177.189,8.276,148.799
C01514=1145.971,282.181,-71.437,-177.185,8.280,148.799
C01515=1145.966,282.430,-71.467,-177.183,8.283,148.800
C01516=1145.962,282.678,-71.497,-177.180,8.286,148.800
C01517=1145.957,282.926,-71.526,-177.177,8.289,148.799
C01518=1145.954,283.174,-71.556,-177.175,8.292,148.800
C01519=1145.949,283.422,-71.586,-177.172,8.296,148.800
C01520=1145.944,283.671,-71.616,-177.169,8.299,148.800
C01521=1145.940,283.919,-71.645,-177.167,8.302,148.800
C01522=1145.936,284.167,-71.675,-177.164,8.305,148.800
C01523=1145.932,284.415,-71.705,-177.161,8.309,148.800
C01524=1145.927,284.664,-71.735,-177.159,8.311,148.800
C01525=1145.923,284.911,-71.765,-177.156,8.316,148.800
C01526=1145.919,285.159,-71.795,-177.153,8.319,148.800
C01527=1145.916,285.408,-71.824,-177.151,8.322,148.800
C01528=1145.911,285.656,-71.855,-177.148,8.325,148.800
C01529=1145.907,285.905,-71.885,-177.146,8.328,148.800
C01530=1145.903,286.152,-71.915,-177.142,8.332,148.800
C01531=1145.898,286.401,-71.945,-177.139,8.335,148.800
C01532=1145.894,286.649,-71.974,-177.137,8.338,148.800
C01533=1145.890,286.897,-72.004,-177.134,8.341,148.800
C01534=1145.884,287.173,-72.038,-177.131,8.345,148.801
C01535=1145.880,287.448,-72.071,-177.129,8.348,148.801
C01536=1145.876,287.723,-72.105,-177.125,8.352,148.801
C01537=1145.871,287.999,-72.138,-177.122,8.356,148.801
C01538=1145.867,288.247,-72.168,-177.120,8.359,148.801
C01539=1145.863,288.495,-72.198,-177.117,8.362,148.801
C01540=1145.859,288.743,-72.228,-177.114,8.365,148.801
C01541=1145.854,288.991,-72.258,-177.112,8.369,148.801
C01542=1145.850,289.239,-72.288,-177.109,8.372,148.801
C01543=1145.845,289.487,-72.319,-177.106,8.375,148.801
C01544=1145.842,289.736,-72.349,-177.104,8.378,148.801
C01545=1145.837,289.984,-72.380,-177.101,8.381,148.801
C01546=1145.833,290.232,-72.409,-177.098,8.385,148.801
C01547=1145.829,290.480,-72.439,-177.096,8.388,148.801
C01548=1145.824,290.728,-72.470,-177.093,8.391,148.801
C01549=1145.820,290.976,-72.499,-177.091,8.395,148.802
C01550=1145.816,291.225,-72.531,-177.087,8.398,148.802
C01551=1145.812,291.472,-72.561,-177.085,8.402,148.802
C01552=1145.808,291.720,-72.591,-177.082,8.405,148.802
C01553=1145.804,291.969,-72.621,-177.080,8.408,148.802
C01554=1145.799,292.216,-72.652,-177.076,8.412,148.802
C01555=1145.796,292.465,-72.682,-177.074,8.415,148.802
C01556=1145.791,292.713,-72.713,-177.071,8.418,148.802
C01557=1145.786,292.961,-72.743,-177.069,8.421,148.802
C01558=1145.782,293.209,-72.773,-177.067,8.424,148.802
C01559=1145.778,293.458,-72.804,-177.063,8.428,148.802
C01560=1145.774,293.705,-72.834,-177.061,8.431,148.802
C01561=1145.770,293.953,-72.865,-177.058,8.434,148.802
C01562=1145.766,294.202,-72.895,-177.056,8.438,148.803
C01563=1145.762,294.450,-72.926,-177.052,8.441,148.803
C01564=1145.757,294.698,-72.957,-177.050,8.445,148.803
C01565=1145.753,294.946,-72.987,-177.047,8.447,148.803
C01566=1145.748,295.194,-73.018,-177.045,8.451,148.803
C01567=1145.745,295.442,-73.048,-177.042,8.455,148.803
C01568=1145.741,295.690,-73.079,-177.039,8.458,148.803
C01569=1145.736,295.938,-73.110,-177.037,8.461,148.803
C01570=1145.733,296.186,-73.140,-177.034,8.464,148.803
C01571=1145.728,296.434,-73.171,-177.031,8.468,148.803
C01572=1145.723,296.682,-73.202,-177.029,8.471,148.803
C01573=1145.720,296.931,-73.232,-177.026,8.474,148.804
C01574=1145.716,297.179,-73.263,-177.024,8.478,148.804
C01575=1145.711,297.427,-73.294,-177.021,8.481,148.804
C01576=1145.707,297.675,-73.325,-177.018,8.485,148.804
C01577=1145.703,297.923,-73.355,-177.015,8.487,148.804
C01578=1145.698,298.171,-73.386,-177.012,8.492,148.804
C01579=1145.694,298.419,-73.417,-177.010,8.495,148.804
C01580=1145.690,298.667,-73.448,-177.007,8.498,148.804
C01581=1145.686,298.915,-73.478,-177.005,8.501,148.804
C01582=1145.682,299.163,-73.510,-177.002,8.505,148.805
C01583=1145.678,299.411,-73.540,-176.999,8.508,148.805
C01584=1145.673,299.659,-73.571,-176.997,8.511,148.805
C01585=1145.670,299.907,-73.602,-176.994,8.514,148.805
C01586=1145.665,300.155,-73.633,-176.991,8.518,148.805
C01587=1145.661,300.403,-73.663,-176.989,8.522,148.805
C01588=1145.657,300.651,-73.695,-176.986,8.525,148.805
C01589=1145.652,300.899,-73.726,-176.983,8.529,148.805
C01590=1145.648,301.148,-73.757,-176.981,8.532,148.806
C01591=1145.644,301.396,-73.787,-176.978,8.535,148.805
C01592=1145.640,301.643,-73.819,-176.975,8.539,148.806
C01593=1145.636,301.892,-73.850,-176.973,8.542,148.806
C01594=1145.631,302.140,-73.881,-176.970,8.545,148.806
C01595=1145.628,302.388,-73.912,-176.968,8.548,148.806
C01596=1145.623,302.636,-73.943,-176.965,8.552,148.806
C01597=1145.619,302.884,-73.974,-176.962,8.555,148.806
C01598=1145.615,303.132,-74.006,-176.960,8.559,148.806
C01599=1145.610,303.379,-74.037,-176.957,8.563,148.807
C01600=1145.606,303.628,-74.068,-176.955,8.566,148.807
C01601=1145.602,303.875,-74.099,-176.952,8.569,148.807
C01602=1145.598,304.124,-74.130,-176.949,8.573,148.807
C01603=1145.593,304.371,-74.162,-176.947,8.576,148.807
C01604=1145.589,304.620,-74.193,-176.944,8.579,148.807
C01605=1145.585,304.867,-74.224,-176.942,8.583,148.807
C01606=1145.581,305.116,-74.255,-176.939,8.587,148.808
C01607=1145.577,305.363,-74.287,-176.936,8.590,148.807
C01608=1145.573,305.612,-74.318,-176.933,8.593,148.808
C01609=1145.569,305.859,-74.350,-176.931,8.597,148.808
C01610=1145.565,306.108,-74.381,-176.928,8.600,148.808
C01611=1145.560,306.355,-74.412,-176.925,8.603,148.808
C01612=1145.556,306.604,-74.443,-176.923,8.607,148.808
C01613=1145.552,306.851,-74.475,-176.920,8.610,148.808
C01614=1145.548,307.100,-74.506,-176.918,8.614,148.809
C01615=1145.544,307.347,-74.537,-176.915,8.617,148.809
C01616=1145.540,307.596,-74.569,-176.912,8.621,148.809
C01617=1145.535,307.843,-74.600,-176.910,8.624,148.809
C01618=1145.532,308.092,-74.632,-176.907,8.628,148.809
C01619=1145.528,308.340,-74.664,-176.904,8.631,148.809
C01620=1145.522,308.588,-74.695,-176.902,8.634,148.809
C01621=1145.519,308.836,-74.727,-176.899,8.638,148.810
C01622=1145.514,309.083,-74.758,-176.897,8.642,148.810
C01623=1145.510,309.332,-74.790,-176.894,8.645,148.810
C01624=1145.506,309.579,-74.821,-176.891,8.649,148.810
C01625=1145.502,309.827,-74.853,-176.889,8.652,148.810
C01626=1145.499,310.075,-74.885,-176.886,8.655,148.810
C01627=1145.493,310.324,-74.916,-176.883,8.659,148.811
C01628=1145.490,310.572,-74.948,-176.881,8.662,148.811
C01629=1145.485,310.819,-74.979,-176.878,8.665,148.811
C01630=1145.482,311.067,-75.011,-176.875,8.670,148.811
C01631=1145.478,311.315,-75.043,-176.873,8.673,148.811
C01632=1145.473,311.563,-75.074,-176.870,8.677,148.811
C01633=1145.469,311.811,-75.106,-176.868,8.680,148.812
C01634=1145.465,312.059,-75.138,-176.865,8.683,148.811
C01635=1145.461,312.307,-75.170,-176.862,8.687,148.812
C01636=1145.456,312.555,-75.202,-176.860,8.690,148.812
C01637=1145.453,312.803,-75.234,-176.857,8.694,148.812
C01638=1145.448,313.081,-75.269,-176.855,8.698,148.812
C01639=1145.443,313.358,-75.306,-176.851,8.702,148.812
C01640=1145.439,313.637,-75.341,-176.848,8.706,148.813
C01641=1145.434,313.914,-75.376,-176.845,8.710,148.813
C01642=1145.429,314.162,-75.408,-176.843,8.713,148.813
C01643=1145.426,314.410,-75.440,-176.840,8.717,148.813
C01644=1145.422,314.658,-75.472,-176.838,8.720,148.813
C01645=1145.417,314.905,-75.504,-176.835,8.724,148.814
C01646=1145.414,315.153,-75.537,-176.832,8.727,148.814
C01647=1145.410,315.401,-75.568,-176.830,8.731,148.814
C01648=1145.405,315.649,-75.601,-176.827,8.735,148.814
C01649=1145.401,315.897,-75.632,-176.824,8.738,148.814
C01650=1145.397,316.145,-75.664,-176.822,8.741,148.814
C01651=1145.393,316.393,-75.697,-176.819,8.745,148.815
C01652=1145.389,316.640,-75.728,-176.817,8.749,148.815
C01653=1145.384,316.889,-75.761,-176.814,8.753,148.815
C01654=1145.381,317.136,-75.793,-176.812,8.756,148.815
C01655=1145.376,317.384,-75.826,-176.809,8.759,148.815
C01656=1145.373,317.633,-75.857,-176.806,8.763,148.815
C01657=1145.368,317.880,-75.889,-176.804,8.766,148.816
C01658=1145.364,318.128,-75.921,-176.801,8.770,148.816
C01659=1145.360,318.376,-75.954,-176.798,8.774,148.816
C01660=1145.356,318.624,-75.986,-176.796,8.777,148.816
C01661=1145.352,318.871,-76.018,-176.793,8.781,148.816
C01662=1145.347,319.120,-76.050,-176.791,8.784,148.817
C01663=1145.344,319.367,-76.083,-176.788,8.788,148.817
C01664=1145.339,319.615,-76.115,-176.786,8.792,148.817
C01665=1145.336,319.863,-76.147,-176.783,8.795,148.817
C01666=1145.332,320.111,-76.180,-176.780,8.799,148.817
C01667=1145.327,320.359,-76.212,-176.778,8.802,148.818
C01668=1145.323,320.606,-76.245,-176.775,8.806,148.818
C01669=1145.319,320.854,-76.277,-176.773,8.809,148.818
C01670=1145.315,321.103,-76.309,-176.770,8.813,148.818
C01671=1145.311,321.350,-76.342,-176.767,8.817,148.818
C01672=1145.307,321.598,-76.374,-176.765,8.820,148.818
C01673=1145.303,321.846,-76.407,-176.762,8.824,148.819
C01674=1145.299,322.093,-76.439,-176.760,8.827,148.819
C01675=1145.295,322.341,-76.472,-176.757,8.831,148.819
C01676=1145.290,322.590,-76.504,-176.754,8.834,148.819
C01677=1145.287,322.837,-76.537,-176.752,8.838,148.819
C01678=1145.282,323.085,-76.569,-176.749,8.842,148.820
C01679=1145.279,323.333,-76.602,-176.747,8.845,148.820
C01680=1145.274,323.581,-76.634,-176.744,8.849,148.820
C01681=1145.270,323.829,-76.668,-176.741,8.852,148.820
C01682=1145.267,324.077,-76.699,-176.739,8.857,148.821
C01683=1145.262,324.325,-76.733,-176.736,8.860,148.821
C01684=1145.258,324.572,-76.766,-176.733,8.864,148.821
C01685=1145.254,324.820,-76.797,-176.731,8.867,148.821
C01686=1145.250,325.067,-76.830,-176.729,8.870,148.821
C01687=1145.245,325.316,-76.863,-176.726,8.874,148.822
C01688=1145.241,325.563,-76.896,-176.724,8.878,148.822
C01689=1145.238,325.811,-76.929,-176.721,8.882,148.822
C01690=1145.234,326.059,-76.962,-176.719,8.885,148.822
C01691=1145.229,326.307,-76.994,-176.716,8.889,148.823
C01692=1145.225,326.555,-77.027,-176.713,8.893,148.823
C01693=1145.222,326.802,-77.060,-176.710,8.897,148.823
C01694=1145.217,327.050,-77.092,-176.708,8.900,148.823
C01695=1145.213,327.298,-77.125,-176.705,8.904,148.823
C01696=1145.209,327.546,-77.159,-176.703,8.907,148.824
C01697=1145.205,327.794,-77.192,-176.700,8.912,148.824
C01698=1145.201,328.041,-77.225,-176.698,8.915,148.824
C01699=1145.197,328.289,-77.257,-176.695,8.918,148.824
C01700=1145.193,328.537,-77.290,-176.692,8.922,148.825
C01701=1145.189,328.785,-77.323,-176.690,8.925,148.825
C01702=1145.185,329.033,-77.356,-176.687,8.929,148.825
C01703=1145.180,329.280,-77.389,-176.685,8.933,148.825
C01704=1145.176,329.528,-77.423,-176.682,8.937,148.826
C01705=1145.172,329.776,-77.456,-176.680,8.940,148.826
C01706=1145.169,330.023,-77.488,-176.677,8.944,148.826
C01707=1145.165,330.271,-77.521,-176.675,8.948,148.826
C01708=1145.161,330.519,-77.555,-176.672,8.952,148.826
C01709=1145.156,330.767,-77.587,-176.669,8.955,148.827
C01710=1145.152,331.015,-77.620,-176.667,8.959,148.827
C01711=1145.148,331.263,-77.654,-176.664,8.962,148.827
C01712=1145.145,331.510,-77.688,-176.662,8.967,148.828
C01713=1145.140,331.758,-77.721,-176.659,8.970,148.828
C01714=1145.136,332.006,-77.754,-176.656,8.974,148.828
C01715=1145.132,332.253,-77.787,-176.654,8.977,148.828
C01716=1145.128,332.501,-77.820,-176.651,8.982,148.828
C01717=1145.124,332.749,-77.853,-176.649,8.985,148.829
C01718=1145.120,332.997,-77.886,-176.646,8.989,148.829
C01719=1145.116,333.244,-77.920,-176.644,8.992,148.829
C01720=1145.111,333.492,-77.953,-176.641,8.997,148.829
C01721=1145.108,333.741,-77.986,-176.639,9.000,148.830
C01722=1145.104,333.988,-78.019,-176.636,9.004,148.830
C01723=1145.100,334.235,-78.053,-176.634,9.007,148.830
C01724=1145.096,334.483,-78.086,-176.631,9.011,148.830
C01725=1145.092,334.731,-78.120,-176.629,9.015,148.831
C01726=1145.088,334.979,-78.153,-176.626,9.019,148.831
C01727=1145.084,335.226,-78.187,-176.623,9.022,148.831
C01728=1145.079,335.474,-78.221,-176.621,9.026,148.831
C01729=1145.075,335.722,-78.254,-176.618,9.030,148.832
C01730=1145.071,335.970,-78.287,-176.616,9.034,148.832
C01731=1145.067,336.217,-78.321,-176.613,9.037,148.832
C01732=1145.063,336.465,-78.354,-176.611,9.041,148.833
C01733=1145.060,336.713,-78.388,-176.608,9.045,148.833
C01734=1145.056,336.960,-78.422,-176.605,9.049,148.833
C01735=1145.052,337.208,-78.455,-176.603,9.053,148.833
C01736=1145.047,337.456,-78.488,-176.600,9.056,148.834
C01737=1145.043,337.703,-78.522,-176.598,9.060,148.834
C01738=1145.039,337.952,-78.556,-176.595,9.064,148.834
C01739=1145.035,338.199,-78.589,-176.593,9.068,148.834
C01740=1145.031,338.446,-78.623,-176.590,9.071,148.835
C01741=1145.027,338.694,-78.657,-176.587,9.075,148.835
C01742=1145.023,338.975,-78.694,-176.585,9.079,148.835
C01743=1145.018,339.255,-78.733,-176.582,9.084,148.836
C01744=1145.014,339.536,-78.771,-176.579,9.088,148.836
C01745=1145.009,339.816,-78.809,-176.576,9.092,148.836
C01746=1145.005,340.063,-78.843,-176.573,9.096,148.836
C01747=1145.000,340.311,-78.877,-176.571,9.100,148.837
C01748=1144.997,340.559,-78.911,-176.568,9.104,148.837
C01749=1144.993,340.807,-78.944,-176.566,9.108,148.837
C01750=1144.988,341.054,-78.979,-176.564,9.111,148.838
C01751=1144.985,341.301,-79.013,-176.561,9.115,148.838
C01752=1144.981,341.550,-79.046,-176.558,9.119,148.838
C01753=1144.977,341.797,-79.081,-176.555,9.123,148.838
C01754=1144.972,342.045,-79.114,-176.554,9.126,148.839
C01755=1144.969,342.293,-79.148,-176.551,9.130,148.839
C01756=1144.965,342.540,-79.183,-176.548,9.135,148.839
C01757=1144.960,342.788,-79.216,-176.546,9.138,148.840
C01758=1144.957,343.036,-79.250,-176.543,9.142,148.840
C01759=1144.953,343.283,-79.284,-176.541,9.146,148.840
C01760=1144.949,343.530,-79.318,-176.538,9.150,148.841
C01761=1144.945,343.779,-79.352,-176.536,9.153,148.841
C01762=1144.941,344.026,-79.386,-176.533,9.157,148.841
C01763=1144.936,344.274,-79.421,-176.530,9.161,148.841
C01764=1144.933,344.521,-79.455,-176.528,9.165,148.842
C01765=1144.929,344.769,-79.488,-176.525,9.169,148.842
C01766=1144.924,345.017,-79.523,-176.523,9.172,148.842
C01767=1144.921,345.264,-79.557,-176.520,9.177,148.843
C01768=1144.916,345.512,-79.591,-176.517,9.181,148.843
C01769=1144.913,345.759,-79.625,-176.515,9.184,148.843
C01770=1144.909,346.007,-79.660,-176.513,9.188,148.843
C01771=1144.904,346.255,-79.693,-176.510,9.192,148.844
C01772=1144.901,346.503,-79.728,-176.508,9.196,148.844
C01773=1144.897,346.750,-79.762,-176.505,9.199,148.844
C01774=1144.893,346.998,-79.797,-176.502,9.203,148.845
C01775=1144.889,347.245,-79.831,-176.500,9.208,148.845
C01776=1144.884,347.493,-79.865,-176.498,9.211,148.845
C01777=1144.880,347.741,-79.900,-176.495,9.215,148.845
C01778=1144.877,347.988,-79.934,-176.493,9.219,148.846
C01779=1144.873,348.236,-79.969,-176.490,9.223,148.846
C01780=1144.869,348.483,-80.002,-176.487,9.227,148.847
C01781=1144.865,348.731,-80.037,-176.485,9.230,148.847
C01782=1144.861,348.978,-80.071,-176.482,9.235,148.847
C01783=1144.857,349.226,-80.106,-176.480,9.239,148.848
C01784=1144.852,349.474,-80.140,-176.477,9.242,148.848
C01785=1144.849,349.721,-80.174,-176.475,9.247,148.848
C01786=1144.845,349.968,-80.210,-176.473,9.250,148.848
C01787=1144.840,350.216,-80.244,-176.470,9.254,148.849
C01788=1144.837,350.464,-80.279,-176.467,9.258,148.849
C01789=1144.833,350.711,-80.313,-176.465,9.262,148.849
C01790=1144.829,350.959,-80.348,-176.462,9.266,148.850
C01791=1144.825,351.207,-80.382,-176.459,9.270,148.850
C01792=1144.821,351.454,-80.417,-176.457,9.274,148.850
C01793=1144.817,351.702,-80.452,-176.455,9.278,148.851
C01794=1144.813,351.949,-80.486,-176.452,9.281,148.851
C01795=1144.809,352.197,-80.521,-176.450,9.285,148.851
C01796=1144.805,352.444,-80.556,-176.447,9.289,148.852
C01797=1144.801,352.692,-80.591,-176.445,9.293,148.852
C01798=1144.797,352.939,-80.625,-176.442,9.297,148.852
C01799=1144.793,353.187,-80.660,-176.439,9.302,148.853
C01800=1144.789,353.434,-80.695,-176.437,9.305,148.853
C01801=1144.785,353.682,-80.730,-176.435,9.309,148.853
C01802=1144.782,353.930,-80.764,-176.432,9.313,148.854
C01803=1144.778,354.177,-80.799,-176.430,9.317,148.854
C01804=1144.774,354.425,-80.834,-176.427,9.321,148.854
C01805=1144.769,354.672,-80.869,-176.424,9.325,148.855
C01806=1144.766,354.920,-80.903,-176.422,9.329,148.855
C01807=1144.762,355.168,-80.938,-176.419,9.333,148.855
C01808=1144.758,355.415,-80.973,-176.417,9.336,148.856
C01809=1144.754,355.663,-81.008,-176.414,9.340,148.856
C01810=1144.750,355.909,-81.043,-176.412,9.345,148.856
C01811=1144.746,356.158,-81.078,-176.409,9.348,148.857
C01812=1144.742,356.405,-81.114,-176.407,9.352,148.857
C01813=1144.738,356.652,-81.148,-176.404,9.356,148.857
C01814=1144.734,356.900,-81.183,-176.402,9.360,148.858
C01815=1144.730,357.148,-81.218,-176.399,9.364,148.858
C01816=1144.726,357.395,-81.253,-176.397,9.368,148.858
C01817=1144.723,357.642,-81.289,-176.394,9.373,148.859
C01818=1144.719,357.890,-81.323,-176.392,9.376,148.859
C01819=1144.714,358.137,-81.359,-176.389,9.380,148.859
C01820=1144.710,358.385,-81.393,-176.386,9.385,148.860
C01821=1144.707,358.633,-81.429,-176.384,9.388,148.860
C01822=1144.702,358.879,-81.464,-176.382,9.392,148.860
C01823=1144.698,359.128,-81.499,-176.379,9.396,148.861
C01824=1144.695,359.375,-81.535,-176.377,9.400,148.861
C01825=1144.691,359.623,-81.570,-176.374,9.404,148.861
C01826=1144.687,359.870,-81.604,-176.371,9.408,148.862
C01827=1144.684,360.117,-81.640,-176.368,9.412,148.862
